BEGIN
	// =============================================================================================================================
	// Purpose: Reditech standard typical for controlling a digital valve (open/close OR 3-way valve)
	// -----------------------------------------------------------------------------------------------------------------------------
	// Date (dd MMM yyyy)   Developer                                   Version Comments/Reason for change
	// ..................   .........                                   ....... ..........................
	// 10 Dec 2018          Bram Verheyen                               08.0    Full review
	// 30 Jan 2019          Matthias De Staelen                         08.1    Outputs can be high in simulation mode
	// =============================================================================================================================

	//============================================================================================
	#b_CfgEnOutpAlwaysOn := #Iw_Cfg.%X1;
	#b_CfgEnFbPos1 := #Iw_Cfg.%X2;
	#b_CfgEnFbPos0 := #Iw_Cfg.%X3;
	#b_CfgSafPosPos1 := #Iw_Cfg.%X4;
	#b_CfgPushToRun := #Iw_Cfg.%X8;
	#b_CfgDisableSim := #Iw_Cfg.%X10;
	#b_CfgStopArea := #Iw_Cfg.%X11;

	//============================================================================================
	#b_DisAlmWrn := #Ib_DisAlmWrn OR #IO_AreaCmd.Alm.Dis OR #b_StaModDis;

	//============================================================================================
	#b_StaSaf := (#Iby_Saf <> 0) AND NOT #b_DisAlmWrn;
	#b_StaIlOn := (#Iby_IlOn <> 0);
	#b_StaIlOff := (#Iby_IlOff <> 0);

	//============================================================================================
	#b_HmiCmdModAut := #IOdi_HmiCmd.%X0;
	#b_HmiCmdModMan := #IOdi_HmiCmd.%X1;
	#b_HmiCmdModDis := #IOdi_HmiCmd.%X2;
	#b_HmiCmdSim := #IOdi_HmiCmd.%X3;
	#b_HmiCmdPos1 := #IOdi_HmiCmd.%X4;
	#b_HmiCmdPos0 := #IOdi_HmiCmd.%X5;
	#b_HmiCmdStp := #IOdi_HmiCmd.%X6;
	#b_HmiCmdRst := #IOdi_HmiCmd.%X7;
	#b_HmiCmdRstActCou := #IOdi_HmiCmd.%X8;

	IF #b_CfgPushToRun THEN
	    #IOdi_HmiCmd := DWORD_TO_DINT(DINT_TO_DWORD(#IOdi_HmiCmd) AND 48);
	ELSE
	    #IOdi_HmiCmd := 0;
	END_IF;

	//============================================================================================
	IF #IO_AreaCmd.Mode.AreaMode THEN
	    #b_ReqAut := #IO_AreaCmd.Mode.Auto;
	    #b_ReqMan := #IO_AreaCmd.Mode.Man;
	    #b_ReqDis := #IO_AreaCmd.Mode.Dis;
	ELSE
	    #b_ReqAut := #b_HmiCmdModAut;
	    #b_ReqMan := #b_HmiCmdModMan;
	    #b_ReqDis := #b_HmiCmdModDis;
	END_IF;

	IF (#b_ReqAut AND NOT #b_ReqMan AND NOT #b_ReqDis) THEN
	    #b_StaModAut := true;
	    #b_StaModMan := false;
	    #b_StaModDis := false;
	END_IF;
	IF (#b_ReqMan AND NOT #b_ReqAut AND NOT #b_ReqDis) THEN
	    #b_StaModAut := false;
	    #b_StaModMan := true;
	    #b_StaModDis := false;
	END_IF;
	IF (#b_ReqDis AND NOT #b_ReqAut AND NOT #b_ReqMan) THEN
	    #b_StaModAut := false;
	    #b_StaModMan := false;
	    #b_StaModDis := true;
	END_IF;

	//============================================================================================
	IF #IO_AreaCmd.Sim.ForceOn OR (#b_HmiCmdSim AND NOT #b_StaSim AND NOT #IO_AreaCmd.Sim.ForceOn AND NOT #IO_AreaCmd.Sim.ForceOff) THEN
	    #b_StaSim := true;
	    #b_HmiCmdSim := false; // reset of command necessary, else simulation will always be reset immediately by following instructions
	END_IF;
	IF #IO_AreaCmd.Sim.ForceOff OR (#b_HmiCmdSim AND #b_StaSim AND NOT #IO_AreaCmd.Sim.ForceOn AND NOT #IO_AreaCmd.Sim.ForceOff) THEN
	    #b_StaSim := false;
	    #b_HmiCmdSim := false;
	END_IF;

	//============================================================================================
	#b_AlActCtn := #Iby_CfgActionAlm.%X0;
	#b_AlActSaf := #Iby_CfgActionAlm.%X1;
	#b_AlActStp := #Iby_CfgActionAlm.%X2;

	#b_CfgAlmActCtn := #b_AlActCtn OR (NOT #b_AlActCtn AND NOT #b_AlActSaf AND NOT #b_AlActStp);
	#b_CfgAlmActSaf := (NOT #b_AlActCtn AND #b_AlActSaf);
	#b_CfgAlmActStp := (NOT #b_AlActCtn AND NOT #b_AlActSaf AND #b_AlActStp);

	//============================================================================================
	IF (#b_ReqPos1 AND NOT #b_FbSimPos1) OR (#b_ReqPos0 AND NOT #b_FbSimPos0) THEN
	    #b_FbSimPos1 := false;
	    #b_FbSimPos0 := false;
	END_IF;
	IF ((#i_TmrFbPos1 <= 1) OR #Ii_ParTFb = 0) AND #b_ReqPos1 THEN
	    #b_FbSimPos1 := true;
	    #b_FbSimPos0 := false;
	END_IF;
	IF ((#i_TmrFbPos0 <= 1) OR #Ii_ParTFb = 0) AND #b_ReqPos0 THEN
	    #b_FbSimPos1 := false;
	    #b_FbSimPos0 := true;
	END_IF;

	//============================================================================================
	#Ob_StaPos1 := (#b_CfgEnFbPos1 AND #Ib_FbPos1 AND NOT #b_StaSim)
	OR (NOT #b_CfgEnFbPos1 AND #b_FbSimPos1)
	OR (#b_StaSim AND #b_FbSimPos1);
	#Ob_StaPos0 := (#b_CfgEnFbPos0 AND #Ib_FbPos0 AND NOT #b_StaSim)
	OR (NOT #b_CfgEnFbPos0 AND #b_FbSimPos0)
	OR (#b_StaSim AND #b_FbSimPos0);

	//============================================================================================
	#b_NoAlm := false;
	#b_RstAlm := #b_HmiCmdRst OR #IO_AreaCmd.Alm.Rst;
	"FC_UTIL_AlmAck"(Ib_CmdAck := #b_RstAlm,
	                 Oi_StaAlm => #i_dummy,
	                 Ob_StaAlm => #b_dummy,
	                 Ob_StaNewAlm => #b_StaAlmNew,
	                 IO_Alm0 := #b_AlmToFb,
	                 IO_Alm1 := #b_AlmIncFb,
	                 IO_Alm2 := #b_AlmIncIl,
	                 IO_Alm3 := #b_NoAlm,
	                 IO_Alm4 := #b_NoAlm,
	                 IO_Alm5 := #b_NoAlm,
	                 IO_Alm6 := #b_NoAlm,
	                 IO_Alm7 := #b_NoAlm,
	                 IO_Alm8 := #b_NoAlm,
	                 IO_Alm9 := #b_NoAlm,
	                 IO_Alm10 := #b_NoAlm,
	                 IO_Alm11 := #b_NoAlm,
	                 IO_Alm12 := #b_NoAlm,
	                 IO_Alm13 := #b_NoAlm,
	                 IO_Alm14 := #b_NoAlm,
	                 IO_Alm15 := #b_NoAlm,
	                 IOi_StaAck := #i_AlmAck);

	//============================================================================================
	IF (#Ii_ParTFb > 0) THEN  // only when time value > 0
	    #FB_UTIL_TON_Del_1(Ii_tValue := #Ii_ParTFb,
	                       Ib_In := (#b_ReqPos1 AND NOT #Ob_StaPos1),
	                       Ii_Base := 1,
	                       Ib_Hold := 0,
	                       Ob_Out => #b_FbErrPos1,
	                       Oi_tmrValue => #i_TmrFbPos1);
	END_IF;

	IF (#Ii_ParTFb > 0) THEN  // only when time value > 0
	    #FB_UTIL_TON_Del_2(Ii_tValue := #Ii_ParTFb,
	                       Ib_In := (#b_ReqPos0 AND NOT #Ob_StaPos0),
	                       Ii_Base := 1,
	                       Ib_Hold := 0,
	                       Ob_Out => #b_FbErrPos0,
	                       Oi_tmrValue => #i_TmrFbPos0);
	END_IF;

	IF ((#b_FbErrPos0 OR #b_FbErrPos1) AND (#Ii_ParTFb > 0)) AND NOT #b_DisAlmWrn THEN
	    #b_AlmToFb := true;
	END_IF;

	//============================================================================================
	IF (#Ii_ParTFb > 0) THEN  // only when time value > 0
	    #FB_UTIL_TON_Del_3(Ii_tValue := #Ii_ParTFb,
	                       Ib_In := (#Ob_StaPos1 AND #Ob_StaPos0),
	                       Ii_Base := 1,
	                       Ib_Hold := 0,
	                       Ob_Out => #b_IncFbErr,
	                       Oi_tmrValue => #i_TmrIncFb);
	END_IF;

	IF (#Ob_StaPos1 AND #Ob_StaPos0 AND #b_IncFbErr) AND NOT #b_DisAlmWrn THEN
	    #b_AlmIncFb := true;
	END_IF;

	//============================================================================================
	IF (#b_StaIlOn AND #b_StaIlOff) AND NOT #b_DisAlmWrn THEN
	    #b_AlmIncIl := true;
	END_IF;
	IF NOT (#b_StaIlOn AND #b_StaIlOff) THEN
	    #b_AlmIncIl := false;
	END_IF;

	//============================================================================================
	#b_StaAlm := #b_AlmToFb OR #b_StaSaf OR #b_AlmIncFb OR #b_AlmIncIl;
	#Ob_Alm := #b_StaAlm;

	//============================================================================================
	#b_CmdAutPos1 := #Ib_AutPos1;
	#b_CmdAutPos0 := #Ib_AutPos0;

	IF #b_StaModAut THEN
	    #b_CmdManPos1 := #b_CmdAutPos1;
	    #b_CmdManPos0 := #b_CmdAutPos0;
	END_IF;

	//============================================================================================
	IF #b_StaModMan AND NOT #b_CfgPushToRun THEN
	    IF (#b_HmiCmdPos1 OR (#b_StaSaf AND #b_CfgSafPosPos1) OR (#b_AlmToFb AND #b_CfgAlmActSaf AND #b_CfgSafPosPos1)) THEN
	        #b_CmdManPos1 := true;
	        #b_CmdManPos0 := false;
	    END_IF;
	    IF (#b_HmiCmdPos0 OR (#b_StaSaf AND NOT #b_CfgSafPosPos1) OR (#b_AlmToFb AND #b_CfgAlmActSaf AND NOT #b_CfgSafPosPos1)) THEN
	        #b_CmdManPos1 := false;
	        #b_CmdManPos0 := true;
	    END_IF;
	    IF #b_HmiCmdStp OR #b_StaAlm OR #b_StaModDis THEN
	        #b_CmdManPos1 := false;
	        #b_CmdManPos0 := false;
	    END_IF;
	END_IF;

	IF #b_StaModMan AND #b_CfgPushToRun THEN
	    #b_CmdManPos1 := ((#b_HmiCmdPos1 AND NOT #b_HmiCmdPos0)
	    OR (#b_StaSaf AND #b_CfgSafPosPos1)
	    OR (#b_AlmToFb AND #b_CfgAlmActSaf AND #b_CfgSafPosPos1)) AND NOT (#b_AlmToFb AND #b_CfgAlmActStp)
	    AND NOT #b_StaModDis;
	    #b_CmdManPos0 := ((#b_HmiCmdPos0 AND NOT #b_HmiCmdPos1)
	    OR (#b_StaSaf AND NOT #b_CfgSafPosPos1)
	    OR (#b_AlmToFb AND #b_CfgAlmActSaf AND NOT #b_CfgSafPosPos1)) AND NOT (#b_AlmToFb AND #b_CfgAlmActStp)
	    AND NOT #b_StaModDis;
	END_IF;

	IF NOT #b_StaModMan OR #b_StaModDis THEN
	    #b_CmdManPos1 := false;
	    #b_CmdManPos0 := false;
	END_IF;




	//============================================================================================
	#b_CmdPos1 := (#b_StaModAut AND #b_CmdAutPos1) OR (#b_StaModMan AND #b_CmdManPos1);
	#b_CmdPos0 := (#b_StaModAut AND #b_CmdAutPos0) OR (#b_StaModMan AND #b_CmdManPos0);

	//============================================================================================
	#b_ReqOutPos1 := (#b_CmdPos1 AND NOT #b_StaAlm AND NOT #b_StaIlOn)
	OR (#b_CmdPos1 AND #b_StaAlm AND NOT #b_StaSaf AND #b_CfgAlmActCtn)
	OR (#b_StaIlOff AND NOT #b_StaAlm AND NOT #b_StaIlOn)
	OR (#b_StaSaf AND #b_CfgSafPosPos1)
	OR (#b_AlmToFb AND #b_CfgAlmActSaf AND #b_CfgSafPosPos1);

	#b_ReqOutPos0 := (#b_CmdPos0 AND NOT #b_StaAlm AND NOT #b_StaIlOff)
	OR (#b_CmdPos0 AND #b_StaAlm AND NOT #b_StaSaf AND #b_CfgAlmActCtn)
	OR (#b_StaIlOn AND NOT #b_StaAlm AND NOT #b_StaIlOff)
	OR (#b_StaSaf AND NOT #b_CfgSafPosPos1)
	OR (#b_AlmToFb AND #b_CfgAlmActSaf AND NOT #b_CfgSafPosPos1);

	#b_ReqPos1 := (#b_ReqOutPos1 AND #b_CfgEnOutpAlwaysOn)
	OR (#b_ReqOutPos1 AND NOT #b_CfgEnOutpAlwaysOn AND NOT #Ob_StaPos1)
	AND NOT #b_StaModDis;
	#b_ReqPos0 := (#b_ReqOutPos0 AND #b_CfgEnOutpAlwaysOn)
	OR (#b_ReqOutPos0 AND NOT #b_CfgEnOutpAlwaysOn AND NOT #Ob_StaPos0)
	AND NOT #b_StaModDis;

	//============================================================================================
	#Ob_Pos0 := #b_ReqPos0;
	#Ob_Pos1 := #b_ReqPos1;
	#Ob_Stp := NOT #Ob_Pos0 AND NOT #Ob_Pos1;

	//============================================================================================
	#Odi_HmiSta.%X0 := #b_StaModAut;
	#Odi_HmiSta.%X1 := #b_StaModMan;
	#Odi_HmiSta.%X2 := #b_StaModDis;
	#Odi_HmiSta.%X3 := #b_StaSim;
	#Odi_HmiSta.%X4 := #b_StaIlOff;
	#Odi_HmiSta.%X5 := #b_StaIlOn;
	#Odi_HmiSta.%X6 := #b_StaSaf;
	#Odi_HmiSta.%X16 := #b_ReqPos1;
	#Odi_HmiSta.%X17 := #b_ReqPos0;
	#Odi_HmiSta.%X18 := #Ob_StaPos1 AND NOT #b_StaAlm;
	#Odi_HmiSta.%X19 := #Ob_StaPos0 AND NOT #b_StaAlm;
	#Odi_HmiSta.%X20 := #b_StaAlm;
	#Odi_HmiSta.%X28 := #IO_AreaCmd.Mode.AreaMode;
	#Odi_HmiSta.%X29 := #b_CfgAlmActCtn;
	#Odi_HmiSta.%X30 := #b_CfgAlmActSaf;
	#Odi_HmiSta.%X31 := #b_CfgAlmActStp;

	#Oi_HMIStaInd.%X0 := 0;
	#Oi_HMIStaInd.%X0 := #b_StaModAut;
	#Oi_HMIStaInd.%X1 := #b_StaModMan;
	#Oi_HMIStaInd.%X2 := #b_StaModDis;
	#Oi_HMIStaInd.%X3 := #b_StaSim;
	#Oi_HMIStaInd.%X4 := #b_StaAlm;
	#Oi_HMIStaInd.%X5 := #Ob_StaPos1 AND NOT #b_StaAlm;
	#Oi_HMIStaInd.%X6 := #Ob_StaPos0 AND NOT #b_StaAlm;

	#I_HmiSta.%X0 := #b_StaModAut;
	#I_HmiSta.%X1 := #b_StaModMan;
	#I_HmiSta.%X2 := #b_StaModDis;
	#I_HmiSta.%X3 := #b_StaSim;
	#I_HmiSta.%X4 := #b_StaIlOn;
	#I_HmiSta.%X5 := #b_StaIlOff;
	#I_HmiSta.%X6 := #Ob_StaPos1;
	#I_HmiSta.%X7 := #Ob_StaPos0;
	#I_HmiSta.%X8 := #b_StaAlm;

	//============================================================================================
	#di_AUX := 0;
	#di_AUX.%X0 := #b_AlmToFb;
	#di_AUX.%X1 := #b_AlmIncFb;
	#di_AUX.%X2 := #b_AlmIncIl;
	#di_AUX.%X8 := #Iby_IlOff.%X0;
	#di_AUX.%X9 := #Iby_IlOff.%X1;
	#di_AUX.%X10 := #Iby_IlOff.%X2;
	#di_AUX.%X11 := #Iby_IlOff.%X3;
	#di_AUX.%X12 := #Iby_IlOff.%X4;
	#di_AUX.%X13 := #Iby_IlOff.%X5;
	#di_AUX.%X14 := #Iby_IlOff.%X6;
	#di_AUX.%X15 := #Iby_IlOff.%X7;
	#di_AUX.%X16 := #Iby_IlOn.%X0;
	#di_AUX.%X17 := #Iby_IlOn.%X1;
	#di_AUX.%X18 := #Iby_IlOn.%X2;
	#di_AUX.%X19 := #Iby_IlOn.%X3;
	#di_AUX.%X20 := #Iby_IlOn.%X4;
	#di_AUX.%X21 := #Iby_IlOn.%X5;
	#di_AUX.%X22 := #Iby_IlOn.%X6;
	#di_AUX.%X23 := #Iby_IlOn.%X7;
	#di_AUX.%X24 := #Iby_Saf.%X0;
	#di_AUX.%X25 := #Iby_Saf.%X1;
	#di_AUX.%X26 := #Iby_Saf.%X2;
	#di_AUX.%X27 := #Iby_Saf.%X3;
	#di_AUX.%X28 := #Iby_Saf.%X4;
	#di_AUX.%X29 := #Iby_Saf.%X5;
	#di_AUX.%X30 := #Iby_Saf.%X6;
	#di_AUX.%X31 := #Iby_Saf.%X7;
	#Odi_HmiAlm := #di_AUX;

	//============================================================================================
	#di_AUX := 0;
	#di_AUX.%X0 := #b_AlmToFb;
	#di_AUX.%X1 := #b_AlmIncFb;
	#di_AUX.%X2 := #b_AlmIncIl;
	#Oi_HmiAlm := DINT_TO_INT(#di_AUX);

	//============================================================================================
	IF #b_StaModDis THEN
	    #IO_AreaFb.Mode.Dis := TRUE;
	END_IF;
	IF #b_StaModMan THEN
	    #IO_AreaFb.Mode.Man := TRUE;
	END_IF;
	IF #b_StaModAut THEN
	    #IO_AreaFb.Mode.Auto := TRUE;
	END_IF;
	IF #b_StaAlm THEN
	    #IO_AreaFb.Alm.Alm := TRUE;
	END_IF;
	IF #b_StaAlmNew THEN
	    #IO_AreaFb.Alm.New := TRUE;
	END_IF;
	IF #b_StaAlm AND #b_CfgStopArea THEN
	    #IO_AreaFb.Alm.StopArea := TRUE;
	END_IF;
	IF #b_StaSim THEN
	    #IO_AreaFb.Sim.Sim := TRUE;
	END_IF;

	//Generating alarm category feedback
	IF #i_Category = 1 AND #b_StaAlm THEN
	    #IO_AreaFb.Alm.Alm_Lvl1 := TRUE;
	END_IF;

	IF #i_Category = 2 AND #b_StaAlm THEN
	    #IO_AreaFb.Alm.Alm_Lvl2 := TRUE;
	END_IF;

	IF #i_Category = 3 AND #b_StaAlm THEN
	    #IO_AreaFb.Alm.Alm_Lvl3 := TRUE;
	END_IF;

	//============================================================================================
	IF (#Ob_Pos0 AND NOT #b_Old_Ob_Pos0) OR (#Ob_Pos1 AND NOT #b_Old_Ob_Pos1) THEN
	    #Odi_ActCouRst := #Odi_ActCouRst + 1;
	    #Odi_ActCouTot := #Odi_ActCouTot + 1;
	END_IF;
	IF #b_HmiCmdRstActCou THEN
	    #Odi_ActCouRst := 0;
	END_IF;
	#b_Old_Ob_Pos0 := #Ob_Pos0;
	#b_Old_Ob_Pos1 := #Ob_Pos1;
END_FUNCTION_BLOCK

FUNCTION_BLOCK "FB_CM_DI"
TITLE = Digital input
{ S7_Optimized_Access := 'FALSE' }
AUTHOR : Reditech
FAMILY : Typical
VERSION : 0.0
//Reditech standard typical for controlling a digital input (switch) inversion is possible, input is delayed
   VAR_INPUT
      Ib_InRaw : Bool;   //  digital input
      Ib_Inv : Bool;   //  invert digital input
      Ii_ParTOn : Int;   //  time delay value ON
      Ii_ParTOff : Int;   //  time delay value OFF
      Ib_EnAlmIfzero : Bool;
      Ib_EnAlmIfOne : Bool;
      Ib_EnWrnIfzero : Bool;
      Ib_EnWrnIfOne : Bool;
      Ib_DisAlmWrn : Bool;
      Iw_Cfg : Word;   //  .0=alarm if out = 0 / .1=alarm if out = 1 / .2=automatic alarm reset / .4 = warning if out =0 / .5 = warning if out =1
   END_VAR

   VAR_OUTPUT
      Ob_Out : Bool;   //  Output value
      Ob_Alm : Bool;   //  general alarm
      Ob_Wrn : Bool;   //  general warning
      Odi_HmiSta : DInt;   //  State bits for HMI
      Odi_HmiAlm : DInt;   //  Alarm bit for HMI
      Oi_HmiAlm : Int;   //  Alarm bit for HMI
   END_VAR

   VAR_IN_OUT
      IOdi_HmiCmd : DInt;   //  Command bits from HMI
      IO_AreaCmd : "UDT_AreaCmd";   //  Command bits from area
      IO_AreaFb : "UDT_AreaFb";   //  Feedback bits to area
   END_VAR

   VAR
      i_TmrOn { ExternalVisible := 'False'} : Int;   //  actual timer value delay ON
      i_TmrOff { ExternalVisible := 'False'} : Int;   //  actual timer value delay OFF
      b_HmiCmdSim { ExternalVisible := 'False'} : Bool;   //  command (toggle) simulation mode
      b_HmiCmdSimValOn { ExternalVisible := 'False'} : Bool;   //  set simulation value on
      b_HmiCmdSimValOff { ExternalVisible := 'False'} : Bool;   //  set simulation value off
      b_HmiCmdRst { ExternalVisible := 'False'} : Bool;   //  reset alarm
      b_StaSim { ExternalVisible := 'False'} : Bool;   //  simulation mode on
      b_StaInRaw { ExternalVisible := 'False'} : Bool;   //  copy of input value
      b_StaAlm { ExternalVisible := 'False'} : Bool;   //  alarm
      b_StaOut { ExternalVisible := 'False'} : Bool;   //  output
      b_StaWrn { ExternalVisible := 'False'} : Bool;   //  warning
      b_CfgAutoReset { ExternalVisible := 'False'} : Bool;   //  automatic alarm reset
      b_CfgStopArea { ExternalVisible := 'False'} : Bool;
      b_Alm { ExternalVisible := 'False'} : Bool;   //  alarm
      b_Wrn { ExternalVisible := 'False'} : Bool;   //  warning
      b_In { ExternalVisible := 'False'} : Bool;   //  auxiliary bit for input value before delays
      b_TOnOut { ExternalVisible := 'False'} : Bool;   //  time delay ON finished
      b_TOffOut { ExternalVisible := 'False'} : Bool;   //  time delay OFF finished
      Fb_UTIL_Ton_Del { ExternalVisible := 'False'} : "FB_UTIL_TON_Sec";
      FB_UTIL_TOF_Del { ExternalVisible := 'False'} : "FB_UTIL_TON_Sec";
      b_DisAlmWrn : Bool;
      b_dummy : Bool;
      i_dummy : Int;
      b_StaAlmNew : Bool;
      b_NoAlm : Bool;
      i_AlmAck : Int;
      b_DisAlmWrn_1 : Bool;
      b_RstAlm : Bool;
      i_Category : Int;   // Device alarm category setting
   END_VAR

   VAR_TEMP
      di_AUX : DInt;   //  auxiliary double word for calculation of state or alarm word to HMI
   END_VAR


BEGIN
	// =========================================================================================================================
	// Purpose: Reditech standard typical for controlling a digital input (switch) inversion is possible, input is delayed
	// -------------------------------------------------------------------------------------------------------------------------
	// Date (dd MMM yyyy)   Developer                                   Version Comments/Reason for change
	// ..................   .........                                   ....... ..........................
	// 18 Dec 2018          Bram Verheyen                               09.0    Full review
	// =========================================================================================================================

	//============================================================================================
	#b_CfgAutoReset := #Iw_Cfg.%X2;
	#b_CfgStopArea := #Iw_Cfg.%X11;

	//============================================================================================
	#b_DisAlmWrn := #Ib_DisAlmWrn OR #IO_AreaCmd.Alm.Dis;

	//============================================================================================
	#b_HmiCmdSim := #IOdi_HmiCmd.%X0;
	#b_HmiCmdSimValOn := #IOdi_HmiCmd.%X1;
	#b_HmiCmdSimValOff := #IOdi_HmiCmd.%X2;
	#b_HmiCmdRst := #IOdi_HmiCmd.%X3;
	#IOdi_HmiCmd := 0;

	//============================================================================================
	IF #IO_AreaCmd.Sim.ForceOn OR (#b_HmiCmdSim AND NOT #b_StaSim AND NOT #IO_AreaCmd.Sim.ForceOn AND NOT #IO_AreaCmd.Sim.ForceOff) THEN
	    #b_StaSim := true;
	    #b_HmiCmdSim := false; // reset of command necessary, else simulation will always be reset immediately by following instructions
	END_IF;
	IF #IO_AreaCmd.Sim.ForceOff OR (#b_HmiCmdSim AND #b_StaSim AND NOT #IO_AreaCmd.Sim.ForceOn AND NOT #IO_AreaCmd.Sim.ForceOff) THEN
	    #b_StaSim := false;
	    #b_HmiCmdSim := false;
	END_IF;

	//============================================================================================
	IF NOT #b_StaSim THEN
	    IF NOT #Ib_Inv THEN
	        #b_In := #Ib_InRaw;
	    ELSE
	        #b_In := NOT #Ib_InRaw;
	    END_IF;
	    #b_StaInRaw := #Ib_InRaw;
	ELSE
	    IF #b_HmiCmdSimValOn THEN
	        #b_In := true;
	    END_IF;
	    IF #b_HmiCmdSimValOff THEN
	        #b_In := false;
	    END_IF;
	    #b_StaInRaw := #b_In;
	END_IF;

	//============================================================================================
	#Fb_UTIL_Ton_Del(Ii_tValue := #Ii_ParTOn,
	                 Ib_In := #b_In AND (#Ib_EnAlmIfOne OR #Ib_EnWrnIfOne) AND NOT #b_DisAlmWrn,
	                 Ii_Base := 1,
	                 Ib_Hold := 0,
	                 Ob_Out => #b_TOnOut,
	                 Oi_tmrValue => #i_TmrOn);

	#FB_UTIL_TOF_Del(Ii_tValue := #Ii_ParTOff,
	                 Ib_In := (NOT #b_In AND (#Ib_EnAlmIfzero OR #Ib_EnWrnIfzero) AND NOT #b_DisAlmWrn),
	                 Ii_Base := 1,
	                 Ib_Hold := 0,
	                 Ob_Out => #b_TOffOut,
	                 Oi_tmrValue => #i_TmrOff);

	#b_StaOut := #b_In;
	//============================================================================================
	#b_NoAlm := false;
	#b_RstAlm := #b_HmiCmdRst OR #IO_AreaCmd.Alm.Rst OR #b_CfgAutoReset;
	"FC_UTIL_AlmAck"(Ib_CmdAck := #b_RstAlm,
	                 Oi_StaAlm => #i_dummy,
	                 Ob_StaAlm => #b_dummy,
	                 Ob_StaNewAlm => #b_StaAlmNew,
	                 IO_Alm0 := #b_Alm,
	                 IO_Alm1 := #b_Wrn,
	                 IO_Alm2 := #b_NoAlm,
	                 IO_Alm3 := #b_NoAlm,
	                 IO_Alm4 := #b_NoAlm,
	                 IO_Alm5 := #b_NoAlm,
	                 IO_Alm6 := #b_NoAlm,
	                 IO_Alm7 := #b_NoAlm,
	                 IO_Alm8 := #b_NoAlm,
	                 IO_Alm9 := #b_NoAlm,
	                 IO_Alm10 := #b_NoAlm,
	                 IO_Alm11 := #b_NoAlm,
	                 IO_Alm12 := #b_NoAlm,
	                 IO_Alm13 := #b_NoAlm,
	                 IO_Alm14 := #b_NoAlm,
	                 IO_Alm15 := #b_NoAlm,
	                 IOi_StaAck := #i_AlmAck);

	//============================================================================================
	IF ((#b_TOnOut AND #Ib_EnAlmIfOne) OR (#b_TOffOut AND #Ib_EnAlmIfzero)) AND NOT #b_DisAlmWrn THEN
	    #b_Alm := true;

	END_IF;

	//============================================================================================
	IF ((#b_TOnOut AND #Ib_EnWrnIfOne) OR (#b_TOffOut AND #Ib_EnWrnIfzero)) AND NOT #b_DisAlmWrn THEN
	    #b_Wrn := true;
	END_IF;

	//============================================================================================
	#b_StaAlm := #b_Alm;
	#Ob_Alm := #b_Alm;

	//============================================================================================
	#b_StaWrn := #b_Wrn;
	#Ob_Wrn := #b_Wrn;

	//============================================================================================
	#Ob_Out := #b_StaOut;

	//============================================================================================
	#Odi_HmiSta.%X0 := #b_StaSim;
	#Odi_HmiSta.%X1 := #b_StaInRaw;
	#Odi_HmiSta.%X16 := #b_StaAlm;
	#Odi_HmiSta.%X17 := #b_StaOut;
	#Odi_HmiSta.%X18 := #b_StaWrn;
	#Odi_HmiSta.%X28 := #IO_AreaCmd.Mode.AreaMode;

	//Sending data to HMI for animated alarm category
	#Odi_HmiSta.%X8 := #i_Category = 1 AND #b_StaAlm;
	#Odi_HmiSta.%X9 := #i_Category = 2 AND #b_StaAlm;
	#Odi_HmiSta.%X19 := #i_Category = 3 AND #b_StaAlm;

	//============================================================================================
	#di_AUX := 0;
	#di_AUX.%X0 := #b_Alm;
	#di_AUX.%X1 := #b_Wrn;
	#Odi_HmiAlm := #di_AUX;
	#Oi_HmiAlm := DINT_TO_INT(#Odi_HmiAlm);

	//============================================================================================
	IF #b_StaAlm THEN
	    #IO_AreaFb.Alm.Alm := TRUE;
	END_IF;
	IF #b_StaWrn THEN
	    #IO_AreaFb.Alm.Wrn := TRUE;
	END_IF;
	IF #b_StaSim THEN
	    #IO_AreaFb.Sim.Sim := TRUE;
	END_IF;
	IF #b_StaAlmNew THEN
	    #IO_AreaFb.Alm.New := TRUE;
	END_IF;
	IF #b_StaAlm AND #b_CfgStopArea THEN
	    #IO_AreaFb.Alm.StopArea := TRUE;
	END_IF;

	//Generating alarm category feedback
	IF #i_Category = 1 AND #b_StaAlm THEN
	    #IO_AreaFb.Alm.Alm_Lvl1 := TRUE;
	END_IF;

	IF #i_Category = 2 AND #b_StaAlm THEN
	    #IO_AreaFb.Alm.Alm_Lvl2 := TRUE;
	END_IF;

	IF #i_Category = 3 AND #b_StaAlm THEN
	    #IO_AreaFb.Alm.Alm_Lvl3 := TRUE;
	END_IF;
END_FUNCTION_BLOCK

FUNCTION_BLOCK "FB_EM_Lvl"
{ S7_Optimized_Access := 'FALSE' }
VERSION : 0.1
   VAR_INPUT
      Ib_RequestEqp { ExternalVisible := 'False'} : Bool;   //  Request equipment Command
      Ib_LvlOff_FirstEqp : Bool;   //  Level switch low low
      Ib_LvlOff_SecondEqp : Bool;   //  Level switch low
      Ib_LvlOn_FirstEqp : Bool;   //  Level switch high
      Ib_LvlOn_SecondEqp : Bool;   //  Level switch High High
      Ib_NrEqp : Bool;   //  Number of equipment used at the same time, 0 = 1 eqp, 1 = 2 eqp
   END_VAR

   VAR_OUTPUT
      Ob_ReqFirstEqp : Bool;   //  Request first equipment
      Ob_ReqSecondEqp : Bool;   //  Request second equipment
   END_VAR

   VAR_IN_OUT
      IO_AreaCmd : "UDT_AreaCmd";   //  Command bits from area
      IO_AreaFb : "UDT_AreaFb";   //  Feedback bits to area
   END_VAR

   VAR
      b_FirstEqpReq : Bool;   //  Request to Equipment 1
      b_SecondEqpReq : Bool;   //  Request to Equipment 2
      b_ReqAut : Bool;   //  Request automatic mode
      b_ReqMan : Bool;
      b_ReqDis : Bool;
   END_VAR


BEGIN
	//not used// =========================================================================================================================
	// Purpose: Reditech standard typical for controlling Pump Toggle manual automatic or semi-automatic
	// -------------------------------------------------------------------------------------------------------------------------
	// Date (dd MMM yyyy)   Developer                                   Version Comments/Reason for change
	// ..................   .........                                   ....... ..........................
	// 16 OCT 2018          Robin Cardinaels                               01      Initial (creation)

	// =========================================================================================================================
	// copy command bits from HMI and reset

	#b_ReqAut := #IO_AreaCmd.Mode.Auto;
	#b_ReqMan := #IO_AreaCmd.Mode.Man;
	#b_ReqDis := #IO_AreaCmd.Mode.Dis;

	IF NOT #b_ReqAut THEN
	    #b_FirstEqpReq := #b_SecondEqpReq := false;
	ELSE
	    IF #Ib_LvlOn_FirstEqp THEN
	        #b_FirstEqpReq := TRUE;
	    END_IF;
	    IF #Ib_LvlOff_FirstEqp THEN
	        #b_FirstEqpReq := FALSE;
	    END_IF;

	    IF #Ib_NrEqp THEN
	        // setting control bits for anaog and digital control.
	        IF #Ib_LvlOn_SecondEqp THEN
	            #b_SecondEqpReq := TRUE;
	        END_IF;
	        IF #Ib_LvlOff_SecondEqp THEN
	            #b_SecondEqpReq := FALSE;
	        END_IF;
	    ELSE
	        #b_SecondEqpReq := false;
	    END_IF;
	END_IF;

	// Set Output For Motor 1
	#Ob_ReqFirstEqp := #Ib_RequestEqp AND #b_FirstEqpReq;

	//Set output for Motor 2
	#Ob_ReqSecondEqp := #Ib_RequestEqp AND #b_SecondEqpReq;

END_FUNCTION_BLOCK

FUNCTION_BLOCK "FB_EM_Toggle_2Eqp"
{ S7_Optimized_Access := 'FALSE' }
VERSION : 0.1
   VAR_INPUT
      Ib_RequestEqp : Bool;   //  Request equipment Command
      Ib_RequestCompEqp : Bool;   //  Request complementary equipment Command
      Ib_ExtToggle : Bool;   //  External Manual toggle
      Ib_Eqp1Fb : Bool;   //  Equipment 1 Running / Open
      Ib_Eqp1Error : Bool;   //  Equipment 1 Error
      Ii_Eqp1OpHours : DInt;   //  Equipment 1 operating hours
      Ib_Eqp2Fb : Bool;   //  Equipment 2 Running / Open
      Ib_Eqp2Error : Bool;   //  Equipment 2 Error
      Ii_Eqp2OpHours : DInt;   //  Equipment 2 Operating hours
      Ii_TBlckStrt : Int;   //  Block simultaniuos Strting time
      Ib_EqpComp : Bool;   //  The equipment complement each other
      Ib_CfgTogRun : Bool;   //  Toggle on running hours
      Ib_EnMan : Bool;   //  Enable manual action
   END_VAR

   VAR_OUTPUT
      Ob_ReqEqp1 : Bool;   //  Request Equipment 1
      Ob_ReqEqp2 : Bool;   //  Request Equipment 2
      Ob_Alm : Bool;   //  General alarm
      Ob_Wrn : Bool;   //  General warning
      Odi_HmiSta : DInt;   //  State bits for HMI
      Odi_HmiAlm : DInt;   //  Alarm bits for HMI
      Oi_HmiAlm : Int;   //  Alarm bits for HMI
   END_VAR

   VAR_IN_OUT
      IOdi_HmiFcnCmd : DInt;   //  .0: automatic/ .1:semiauto/ .2:manual
      IOdi_HmiCmd : DInt;   //  Command bits from HMI
      IO_AreaCmd : "UDT_AreaCmd";   //  Command bits from area
      IO_AreaFb : "UDT_AreaFb";   //  Feedback bits to area
   END_VAR

   VAR
      b_HmiCmdModAut : Bool;   //  HMI Command Automatic mode
      b_HmiCmdRst : Bool;   //  HMI Command Reset
      b_HmiCmdModMan : Bool;   //  HMI Command Manual mode
      b_HmiCmdModDis : Bool;   //  HMI Command disabled Mode
      b_HmiCmdFrcEqp1First : Bool;   //  HMI Command Force equipment 1 first
      b_HmiCmdFrcEqp2First : Bool;   //  HMI Command Force equipment 2 first
      b_HmiFcnCmdAuto : Bool := TRUE;   //  HMI Functional command automatic mode
      b_HmiFcnCmdManual : Bool;   //  HMI Functional command manual mode
      b_HmiStaAlm : Bool;   //  HMI Status alarm
      b_HmiStaModAut : Bool;   //  HMI status Ready
      b_HmiStaModMan : Bool;   //  HMI Status Running
      b_HmiStaModDis : Bool;   //  HMI status Preference Eqp
      b_HmiStaFcnAuto : Bool := TRUE;   //  HMI Status Fuction auto switch enabled
      b_HmiStaFcnMan : Bool;   //  HMI Status Fuction manual switch enabled
      b_HmiStaOff : Bool;   //  HMI Status OFF
      b_HmiStaReady : Bool;   //  HMI Status Ready
      b_HmiStaRunning : Bool;   //  HMI Status Running
      b_HmiStaPref1 : Bool;   //  HMI Status Preferd Eqp 1
      b_HmiStaWrn : Bool;   //  HMI Status equipment not ready
      b_HmiStaPref2 : Bool;   //  HMI Status Preferd Eqp 2
      b_HmiStaAreaMode : Bool;   //  HMI Status Area Mode
      b_HmiAlmAlm : Bool;   //  General Alarm
      b_HmiWrnEquip : Bool;   //  Equipment not available
      b_Eqp2First : Bool;   //  Toggle bit for Equipment selection; 1 = Eqp 2 first, 0 = eqp1 first
      b_Temp1 : Bool;   //  Equipments running for RE
      b_PrevTemp1 : Bool;   //  prev equipments running for RE
      b_Temp2 : Bool;   //  command manual toggle for RE
      b_PrevTemp2 : Bool;   //  prev command manual toggle for RE
      FB_UTIL_TON_Del_1 : "FB_UTIL_TON_Sec";   //  Timer block Strt to prevent simultainious Strting
      b_BlckStrt : Bool;   //  Block Strt to prevent Strting simultainous
      b_helpReady : Bool;   //  Help bit for status ready
      b_ReqAut : Bool;   //  Request automatic mode
      b_ReqMan : Bool;
      b_ReqDis : Bool;
   END_VAR

   VAR_TEMP
      di_AUX : DInt;   //  auxiliary double word for calculation of state or alarm word to HMI
   END_VAR


BEGIN
	//not used// =========================================================================================================================
	// Purpose: Reditech standard typical for controlling Pump Toggle manual automatic or semi-automatic
	// -------------------------------------------------------------------------------------------------------------------------
	// Date (dd MMM yyyy)   Developer                                   Version Comments/Reason for change
	// ..................   .........                                   ....... ..........................
	// 16 OCT 2018          Robin Cardinaels                               01      Initial (creation)
	// 15 Jan 2019          Robin Cardinaels                               02      Review
	// =========================================================================================================================
	// copy command bits from HMI and reset
	#b_HmiCmdModAut := #IOdi_HmiCmd.%X0;
	#b_HmiCmdModMan := #IOdi_HmiCmd.%X1;
	#b_HmiCmdRst := #IOdi_HmiCmd.%X3;


	#IOdi_HmiCmd := 0;

	// Copy of Function Command bits
	#b_HmiFcnCmdAuto := #IOdi_HmiFcnCmd.%X0;
	#b_HmiFcnCmdManual := #IOdi_HmiFcnCmd.%X2;
	#b_HmiCmdFrcEqp1First := #IOdi_HmiFcnCmd.%X4;
	#b_HmiCmdFrcEqp2First := #IOdi_HmiFcnCmd.%X5;
	#IOdi_HmiFcnCmd := 0;

	IF #b_HmiStaAreaMode THEN
	    #b_ReqAut := #IO_AreaCmd.Mode.Auto;
	    #b_ReqMan := #IO_AreaCmd.Mode.Man;
	    #b_ReqDis := #IO_AreaCmd.Mode.Dis;
	ELSE
	    #b_ReqAut := #b_HmiCmdModAut AND NOT #b_HmiStaAlm;
	    #b_ReqMan := #b_HmiCmdModMan OR (#b_HmiStaAlm AND NOT #b_HmiStaModDis);
	    #b_ReqDis := #b_HmiCmdModDis;
	END_IF;

	IF (#b_ReqAut AND NOT #b_ReqMan AND NOT #b_ReqDis) THEN
	    #b_HmiStaModAut := true;
	    #b_HmiStaModMan := false;
	    #b_HmiStaModDis := false;
	END_IF;
	IF (#b_ReqMan AND NOT #b_ReqAut AND NOT #b_ReqDis) THEN
	    #b_HmiStaModAut := false;
	    #b_HmiStaModMan := true;
	    #b_HmiStaModDis := false;
	END_IF;
	IF (#b_ReqDis AND NOT #b_ReqAut AND NOT #b_ReqMan) THEN
	    #b_HmiStaModAut := false;
	    #b_HmiStaModMan := false;
	    #b_HmiStaModDis := true;
	END_IF;

	// copy Function modes to status bits
	IF #b_HmiFcnCmdAuto THEN
	    #b_HmiStaFcnAuto := true;
	    #b_HmiStaFcnMan := false;
	END_IF;
	IF #b_HmiFcnCmdManual AND #Ib_EnMan THEN
	    #b_HmiStaFcnAuto := false;
	    #b_HmiStaFcnMan := true;
	END_IF;

	#b_PrevTemp1 := #b_Temp1;// temperoraty variable to get rising edge
	#b_Temp1 := (#Ob_ReqEqp1) OR (#Ob_ReqEqp2);

	// IF auto mode selected check operating hours every Time both motors are not running
	IF (NOT #b_Temp1 AND #b_PrevTemp1) AND (#b_HmiStaFcnAuto AND NOT #b_HmiStaFcnMan) THEN
	    IF #Ib_CfgTogRun THEN //equipment with the lowest operating hours will Strt if Configurated
	        #b_Eqp2First := #Ii_Eqp2OpHours < #Ii_Eqp1OpHours; // reset toggle if equipment1 operating hours <= equipment2 operating hours
	    ELSE
	        #b_Eqp2First := NOT #b_Eqp2First;
	    END_IF;
	END_IF;
	#b_PrevTemp2 := #b_Temp2; // prev value of manual toggle command for RE
	#b_Temp2 := #Ib_ExtToggle; // manual toggle command
	//toggle equipments if manual toggle requested (hmi or external) and manual toggle configurated
	IF (#b_Temp2 AND NOT #b_PrevTemp2) AND (#b_HmiStaFcnAuto AND NOT #b_HmiStaFcnMan) THEN
	    #b_Eqp2First := NOT #b_Eqp2First;
	END_IF;

	// set equipment 2 actif if equipment 1 not available
	IF (#Ib_Eqp1Error OR #b_HmiCmdFrcEqp2First) AND NOT #Ib_Eqp2Error THEN
	    #b_Eqp2First := TRUE;
	END_IF;
	// set equipment 1 actif if equipment 2 not available
	IF (#Ib_Eqp2Error OR #b_HmiCmdFrcEqp1First) AND NOT #Ib_Eqp1Error THEN
	    #b_Eqp2First := FALSE;
	END_IF;

	// Set Output of FB
	// Set Output For equipment 1
	#Ob_ReqEqp1 := NOT #Ib_Eqp1Error AND (((#Ib_RequestEqp AND NOT #b_Eqp2First) AND (#b_BlckStrt OR #Ob_ReqEqp1) OR (#Ib_RequestCompEqp AND NOT #b_BlckStrt)) AND #Ib_EqpComp)
	OR (NOT #Ib_EqpComp AND #Ib_RequestEqp AND NOT #b_Eqp2First);

	//Set output for equipment 2
	#Ob_ReqEqp2 := NOT #Ib_Eqp2Error AND (((#Ib_RequestEqp AND #b_Eqp2First) AND (#b_BlckStrt OR #Ob_ReqEqp2) OR (#Ib_RequestCompEqp AND NOT #b_BlckStrt)) AND #Ib_EqpComp)
	OR (NOT #Ib_EqpComp AND #Ib_RequestEqp AND #b_Eqp2First);

	// timer to prevent simultanius Strting
	#FB_UTIL_TON_Del_1(Ii_tValue := #Ii_TBlckStrt,
	                   Ib_In := #Ob_ReqEqp1 OR #Ob_ReqEqp2,
	                   Ii_Base := 1,
	                   Ib_Hold := 0);

	// enable starting again
	#b_BlckStrt := NOT #FB_UTIL_TON_Del_1.Ob_Out;

	// HMI Status
	// Status Ready
	#b_helpReady := ((NOT #Ib_Eqp1Error OR NOT #Ib_Eqp2Error) AND NOT #Ib_EqpComp) OR //help bit ready if one equipment availeble in 1+1
	(NOT #Ib_Eqp1Error AND NOT #Ib_Eqp2Error); // or both equipments available
	#b_HmiStaReady := #b_helpReady AND NOT #b_HmiStaRunning;
	//Status Running
	#b_HmiStaRunning := #b_helpReady AND (#Ib_Eqp1Fb OR #Ib_Eqp2Fb);
	//Status OFF
	#b_HmiStaOff := NOT #b_HmiStaReady AND NOT #b_HmiStaRunning;
	// Show Prefferd Pump
	#b_HmiStaPref1 := NOT #b_Eqp2First;
	#b_HmiStaPref2 := #b_Eqp2First;
	//Wrning when motor not available
	#b_HmiWrnEquip := (#Ib_Eqp1Error OR #Ib_Eqp2Error) AND NOT #b_HmiAlmAlm;
	// status warning
	#b_HmiStaWrn := #b_HmiWrnEquip;
	#Ob_Wrn := #b_HmiWrnEquip;
	//Alarm when both pumps ar inavailable // auto reset if equipment is available
	#b_HmiAlmAlm := #Ib_Eqp1Error AND #Ib_Eqp2Error;

	// general alarm
	#b_HmiStaAlm := #b_HmiAlmAlm;
	#Ob_Alm := #b_HmiAlmAlm;

	// copy state bits into double word for HMI
	#di_AUX := 0;

	#di_AUX.%X0 := #b_HmiStaModAut;
	#di_AUX.%X1 := #b_HmiStaModMan;
	#di_AUX.%X2 := #b_HmiStaModDis;
	#di_AUX.%X8 := #b_HmiStaFcnAuto;

	#di_AUX.%X10 := #b_HmiStaFcnMan;
	#di_AUX.%X15 := #b_HmiStaOff;
	#di_AUX.%X16 := #b_HmiStaAlm;
	#di_AUX.%X21 := #b_HmiStaReady;
	#di_AUX.%X22 := #b_HmiStaRunning;
	#di_AUX.%X23 := #b_HmiStaPref1;
	#di_AUX.%X24 := #b_HmiStaWrn;
	#di_AUX.%X25 := #b_HmiStaPref2;
	#di_AUX.%X29 := #b_HmiStaAreaMode;

	#Odi_HmiSta := #di_AUX;

	// copy alarm bits into double word for HMI
	#di_AUX := 0;
	#di_AUX.%X0 := #b_HmiAlmAlm;
	#di_AUX.%X1 := #b_HmiWrnEquip;

	#Odi_HmiAlm := #di_AUX;
	#Oi_HmiAlm := DINT_TO_INT(#di_AUX);

	// Set feedback bits to area
	// #IO_AreaFb.Mode.Dis := #b_HmiStaModDis;
	// #IO_AreaFb.Mode.Man := #b_HmiStaModMan;
	// #IO_AreaFb.Mode.Auto := #b_HmiStaModAut;
	// #IO_AreaFb.Alm.Alm := #b_HmiStaAlm;
	// #IO_AreaFb.Alm.Wrn := #b_HmiStaWrn;
END_FUNCTION_BLOCK

FUNCTION_BLOCK "FB_UM_Mode"
{ S7_Optimized_Access := 'FALSE' }
VERSION : 0.1
   VAR_INPUT
      Ib_CmdRstAlm : Bool;
      Ib_CmdGenRelease : Bool;
      Ib_CmdRstRelease : Bool;
      Ib_CmdGenDis : Bool;
      Ib_AreaStopped : Bool;
      Ib_AreaCmdMode : Bool;
      Ib_SimForceOn : Bool;
      Ib_SimForceOff : Bool;
      Ib_DCSPermissive : Bool;
   END_VAR

   VAR_OUTPUT
      Odi_HmiSta : DInt;
      Ou_AreaCmd : "UDT_AreaCmd";
      Ob_StaExecute : Bool;
      Ob_StaAlm : Bool;
      Ob_StaWrn : Bool;
      Ob_StaRstAlm : Bool;
      Ob_StaSim : Bool;
      Ou_CurrentMode : "UDT_PML_Mode";
   END_VAR

   VAR_IN_OUT
      IOdi_HmiCmd : DInt;
      IOu_AreaFb : "UDT_AreaFb";
      Ib_CmdGenMan : Bool;
      IOw_DCSCmd : Word;
   END_VAR

   VAR
      PML_ModeManager : "FB_PML_ModeManager";
      b_HmiCmdStart : Bool;
      b_HmiCmdModSimOn : Bool;
      b_HmiCmdModMan : Bool;
      b_HmiCmdModDis : Bool;
      b_HmiCmdModAuto : Bool;
      b_HmiCmdRstAlm : Bool;
      b_HmiCmdModSimOff : Bool;
      b_HmiCmdStop : Bool;
      b_StaRun : Bool;
      AreaFb : "UDT_AreaFb";
      AreaCmd : "UDT_AreaCmd";
      b_StaSim { ExternalAccessible := 'False'; ExternalVisible := 'False'; ExternalWritable := 'False'} : Bool;
      StaAreaFb : "UDT_AreaFb";
      b_StaAlm_Lvl1 { S7_SetPoint := 'True'} : Bool;
      b_StaAlm_Lvl2 : Bool;
      b_StaAlm_Lvl3 : Bool;
      I_HmiSta : Word;
   END_VAR


BEGIN
	// =========================================================================================================================
	// Purpose: Reditech standard typical for handling mode transition with the Reditech's standard PackML ModeManager
	// -------------------------------------------------------------------------------------------------------------------------
	// Date (dd MMM yyyy)   Developer                                   Version Comments/Reason for change
	// ..................   .........                                   ....... ..........................
	// 19 NOV 2018          Gijs van Hal                                01      Initial (creation)
	// 20 OCT 2020          Ivan Galhardoni                             02      Implemented manual mode external request input
	// 12 DEC 2020          Ivan Galhardoni                             03      Implemented alarm level animated signaling
	// =========================================================================================================================

	// Copy HMI commands
	#b_HmiCmdModMan := (#IOdi_HmiCmd.%X0 OR (#IOw_DCSCmd.%X1 AND #Ib_DCSPermissive)) OR #Ib_CmdGenMan AND NOT #Ib_CmdGenDis;
	#b_HmiCmdModDis := ((#IOdi_HmiCmd.%X1  OR (#IOw_DCSCmd.%X2 AND #Ib_DCSPermissive)) OR #Ib_CmdGenDis) AND NOT #Ib_CmdGenMan;
	#b_HmiCmdModAuto := (#IOdi_HmiCmd.%X2 OR (#IOw_DCSCmd.%X0 AND #Ib_DCSPermissive)) AND NOT #Ib_CmdGenDis;
	#b_HmiCmdModSimOn := #IOdi_HmiCmd.%X3;
	#b_HmiCmdModSimOff := #IOdi_HmiCmd.%X4;
	#b_HmiCmdStart := (#IOdi_HmiCmd.%X5 OR (#IOw_DCSCmd.%X3 AND #Ib_DCSPermissive)) AND #PML_ModeManager.Ou_ModeCurrent.Production;
	#b_HmiCmdStop := (#IOdi_HmiCmd.%X6 OR (#IOw_DCSCmd.%X4 AND #Ib_DCSPermissive)) OR #Ib_CmdGenDis;
	#b_HmiCmdRstAlm := #IOdi_HmiCmd.%X7;
	#IOdi_HmiCmd := 0;
	#IOw_DCSCmd := 0;


	// Mode change only possible if area is stopped
	IF #Ib_AreaStopped THEN
	    // Set Iu_CmdMode for ModeManager
	    #PML_ModeManager.Iu_CmdMode.Manual := #b_HmiCmdModMan;
	    #PML_ModeManager.Iu_CmdMode.Disabled := #b_HmiCmdModDis;
	    #PML_ModeManager.Iu_CmdMode.Production := #b_HmiCmdModAuto;

	    // If Mode command is given, mode change request = true
	    IF (#b_HmiCmdModMan OR #b_HmiCmdModDis OR #b_HmiCmdModAuto) THEN
	        #PML_ModeManager.IOb_CmdModeChangeRequest := TRUE;
	    ELSE
	        #PML_ModeManager.IOb_CmdModeChangeRequest := FALSE;
	    END_IF;

	END_IF;

	// Current state
	IF #b_StaRun THEN
	    #PML_ModeManager.Idi_StateCurrent := 6; // Execute State
	ELSE
	    #PML_ModeManager.Idi_StateCurrent := 2; // Stopped State
	END_IF;

	#PML_ModeManager();

	// If Cmd Simulation mode
	IF (#b_HmiCmdModSimOn) THEN
	    #b_StaSim := TRUE;
	ELSIF (#b_HmiCmdModSimOff) THEN
	    #b_StaSim := FALSE;
	END_IF;

	// If start and stop area
	IF (#b_HmiCmdStart) THEN
	    #b_StaRun := TRUE;
	END_IF;
	IF (#b_HmiCmdStop OR #Ib_CmdRstRelease OR #Ib_CmdGenMan) THEN
	    #b_StaRun := FALSE;
	END_IF;


	// Write outputs
	#Ob_StaExecute := #Ib_CmdGenRelease AND #b_StaRun;
	#Ob_StaAlm := #IOu_AreaFb.Alm.Alm;
	#Ob_StaWrn := #IOu_AreaFb.Alm.Wrn;
	#Ob_StaRstAlm := #Ib_CmdRstAlm OR #b_HmiCmdRstAlm;
	#Ob_StaSim := #b_StaSim;
	#b_StaAlm_Lvl1 := #IOu_AreaFb.Alm.Alm_Lvl1;
	#b_StaAlm_Lvl2 := #IOu_AreaFb.Alm.Alm_Lvl2;
	#b_StaAlm_Lvl3 := #IOu_AreaFb.Alm.Alm_Lvl3;

	// Area commands
	#Ou_AreaCmd.Alm.Rst := #Ib_CmdRstAlm OR #b_HmiCmdRstAlm;
	#Ou_AreaCmd.Mode.Man := #PML_ModeManager.Ou_ModeCurrent.Manual;
	#Ou_AreaCmd.Mode.Dis := #PML_ModeManager.Ou_ModeCurrent.Disabled;
	#Ou_AreaCmd.Mode.Auto := #PML_ModeManager.Ou_ModeCurrent.Production;
	#Ou_AreaCmd.Sim.ForceOff := #Ib_SimForceOff;
	#Ou_AreaCmd.Sim.ForceOn := #Ib_SimForceOn;
	#Ou_AreaCmd.Mode.AreaMode := #Ib_AreaCmdMode;

	// Write Current Mode UDT to output.
	#Ou_CurrentMode.Production := #PML_ModeManager.Ou_ModeCurrent.Production;
	#Ou_CurrentMode.Manual := #PML_ModeManager.Ou_ModeCurrent.Manual;
	#Ou_CurrentMode.Disabled := #PML_ModeManager.Ou_ModeCurrent.Disabled;

	// Status Area feedback
	#StaAreaFb.Alm.Alm := #IOu_AreaFb.Alm.Alm;
	#StaAreaFb.Alm.Wrn := #IOu_AreaFb.Alm.Wrn;
	#StaAreaFb.Alm.New := #IOu_AreaFb.Alm.New;
	#StaAreaFb.Alm.StopArea := #IOu_AreaFb.Alm.StopArea;

	// Reset Area feedback
	#IOu_AreaFb.Alm.Alm := FALSE;
	#IOu_AreaFb.Alm.Wrn := FALSE;
	#IOu_AreaFb.Alm.New := FALSE;
	#IOu_AreaFb.Alm.StopArea := FALSE;
	#IOu_AreaFb.Alm.Alm_Lvl1 := FALSE;
	#IOu_AreaFb.Alm.Alm_Lvl2 := FALSE;
	#IOu_AreaFb.Alm.Alm_Lvl3 := FALSE;


	// Copy state bits into double word for HMI
	#Odi_HmiSta.%X0 := #PML_ModeManager.Ou_ModeCurrent.Manual;
	#Odi_HmiSta.%X1 := #PML_ModeManager.Ou_ModeCurrent.Disabled;
	#Odi_HmiSta.%X2 := #PML_ModeManager.Ou_ModeCurrent.Production;
	#Odi_HmiSta.%X3 := #Ob_StaSim;
	#Odi_HmiSta.%X4 := #Ob_StaAlm;
	#Odi_HmiSta.%X5 := #Ob_StaWrn;
	#Odi_HmiSta.%X6 := #b_StaRun;
	#Odi_HmiSta.%X7 := #Ib_AreaStopped;
	#Odi_HmiSta.%X8 := #b_StaAlm_Lvl1;    //Animated Lvl1 area alarm status
	#Odi_HmiSta.%X9 := #b_StaAlm_Lvl2;    //Animated Lvl2 area alarm status
	#Odi_HmiSta.%X10 := #b_StaAlm_Lvl3;   //Animated Lvl3 area alarm status


	// Copy state bits into word for HMI
	#I_HmiSta.%X0 := #PML_ModeManager.Ou_ModeCurrent.Production;
	#I_HmiSta.%X1 := #PML_ModeManager.Ou_ModeCurrent.Manual;
	#I_HmiSta.%X2 := #PML_ModeManager.Ou_ModeCurrent.Disabled;
	#I_HmiSta.%X3 := #b_StaRun;
	#I_HmiSta.%X4 := NOT #b_StaRun;
	#I_HmiSta.%X7 := #Ib_AreaStopped;
	#I_HmiSta.%X8 := #Ob_StaAlm;
	#I_HmiSta.%X9 := #Ob_StaWrn;



END_FUNCTION_BLOCK

FUNCTION_BLOCK "FB_CM_AXV"
TITLE = Analog valve
{ S7_Optimized_Access := 'FALSE' }
AUTHOR : Reditech
FAMILY : Typical
VERSION : 0.0
//Reditech standard typical for controlling an analog valve
   VAR_INPUT
      Ib_FbPosOpn : Bool := FALSE;   //  feedback position open (failsafe : 0=open)
      Ib_FbPosCls : Bool := FALSE;   //  feedback position closed (failsafe : 0=closed)
      Ir_ActPos : Real;   //  Actual valve position (measurement)
      Ir_ParAutSp : Real;   //  automatic setpoint
      Ir_ParMaxPos : Real := 100.0;   //  Maximum position value
      Ir_ParMinPos : Real;   //  Minimum position value
      Ir_ParCtlDev : Real := 1.0;   //  Control deviation (for digital output and feedback OK)
      Ir_ParSafPos : Real;   //  Safety position
      Ir_ParMaxRaw : Real;   //  Max value for analogue output mode
      Ir_ParMinRaw : Real;   //  Min value for analogue output mode
      Ii_ParTO : Int := 5;   //  time out value for feedback monitoring
      Iby_Saf : Byte := 16#00;   //  8 safety bits : 1=error
      Iby_IlOn : Byte;   //  8 interlock bits : 1 prevents Pos1/opening
      Iby_IlOff { ExternalVisible := 'False'} : Byte;   //  8 interlock bits : 1 prevents Pos0/closing
      Ib_Pls1S : Bool;
      Ib_DisAlmWrn : Bool;
      Iw_Cfg : Word := 16#0000;   //  .0=analog pos present / .1=digital pos present
   END_VAR

   VAR_OUTPUT
      Or_SpOut : Real;   //  Control output
      Ow_SpRaw : Word;   //  Control output recalculated for analog output node
      Ob_Opn : Bool;   //  control output open
      Ob_Cls : Bool;   //  control output close
      Ob_PosOk : Bool;   //  Position reached
      Ob_Alm : Bool;   //  general alarm
      Ob_StaOpn : Bool;   //  Status in position 1
      Ob_StaCls : Bool;   //  Status in position 0
      Or_StaPos : Real;
      Odi_HmiSta : DInt;   //  State bits for HMI
      Oi_HmiAlm : Int;
      Odi_HmiAlm : DInt;   //  Alarm bit for HMI
   END_VAR

   VAR_IN_OUT
      IOr_ManSP : Real;   //  manual setpoint
      IOr_SimPos : Real := 0.0;   //  Simulated position
      IOdi_HmiCmd : DInt := 0;   //  Command bits from HMI
      IO_AreaCmd : "UDT_AreaCmd";   //  Command bits from area
      IO_AreaFb : "UDT_AreaFb";   //  Feedback bits to area
   END_VAR

   VAR
      i_TmrFbPos : Int;   //  timer feedback control
      b_HmiCmdModAut { ExternalAccessible := 'False'; ExternalVisible := 'False'; ExternalWritable := 'False'} : Bool;   //  command change mode to AUTO
      b_HmiCmdModMan { ExternalAccessible := 'False'; ExternalVisible := 'False'; ExternalWritable := 'False'} : Bool;   //  command change mode to MANUAL
      b_HmiCmdModDis { ExternalAccessible := 'False'; ExternalVisible := 'False'; ExternalWritable := 'False'} : Bool;   //  command change mode to DISABLED
      b_HmiCmdSim { ExternalAccessible := 'False'; ExternalVisible := 'False'; ExternalWritable := 'False'} : Bool;   //  toggle simulation mode
      b_HmiCmdRst { ExternalAccessible := 'False'; ExternalVisible := 'False'; ExternalWritable := 'False'} : Bool;   //  reset alarms
      b_StaModAut { ExternalAccessible := 'False'; ExternalVisible := 'False'; ExternalWritable := 'False'} : Bool;   //  state AUTOMATIC
      b_StaModMan { ExternalAccessible := 'False'; ExternalVisible := 'False'; ExternalWritable := 'False'} : Bool := TRUE;   //  state MANUAL
      b_StaModDis { ExternalAccessible := 'False'; ExternalVisible := 'False'; ExternalWritable := 'False'} : Bool;   //  state DISABLED
      b_StaSim { ExternalAccessible := 'False'; ExternalVisible := 'False'; ExternalWritable := 'False'} : Bool;   //  state simulation ON
      b_StaIlOff { ExternalAccessible := 'False'; ExternalVisible := 'False'; ExternalWritable := 'False'} : Bool;   //  state interlock OFF : 1 = interlocked (prevents closing)
      b_StaIlOn { ExternalAccessible := 'False'; ExternalVisible := 'False'; ExternalWritable := 'False'} : Bool;   //  state interlock ON : 1 = interlocked (prevents opening)
      b_StaSaf { ExternalAccessible := 'False'; ExternalVisible := 'False'; ExternalWritable := 'False'} : Bool;   //  state safety : 1 = error (valve to safety position)
      b_ReqOpn { ExternalAccessible := 'False'; ExternalVisible := 'False'; ExternalWritable := 'False'} : Bool;   //  output command open
      b_ReqCls { ExternalAccessible := 'False'; ExternalVisible := 'False'; ExternalWritable := 'False'} : Bool;   //  output command close
      b_StaPosOk { ExternalAccessible := 'False'; ExternalVisible := 'False'; ExternalWritable := 'False'} : Bool;   //  position (setpoint) reached
      b_StaAlm { ExternalAccessible := 'False'; ExternalVisible := 'False'; ExternalWritable := 'False'} : Bool;   //  general alarm
      b_CfgAnaPosPres { ExternalAccessible := 'False'; ExternalVisible := 'False'; ExternalWritable := 'False'} : Bool;   //  configuration : analog position feedback present
      b_CfgDigPosPres { ExternalAccessible := 'False'; ExternalVisible := 'False'; ExternalWritable := 'False'} : Bool;   //  configuration : digital limit positions present (min and max)
      b_CfgHldMod { ExternalAccessible := 'False'; ExternalVisible := 'False'; ExternalWritable := 'False'} : Bool;
      b_CfgDisableSim { ExternalAccessible := 'False'; ExternalVisible := 'False'; ExternalWritable := 'False'} : Bool;
      b_CfgStopArea { ExternalAccessible := 'False'; ExternalVisible := 'False'; ExternalWritable := 'False'} : Bool;
      b_AlmToFb { ExternalAccessible := 'False'; ExternalVisible := 'False'; ExternalWritable := 'False'} : Bool;   //  alarm time out feedback
      b_AlmFbInc { ExternalAccessible := 'False'; ExternalVisible := 'False'; ExternalWritable := 'False'} : Bool;   //  alarm inconsistent feedbacks (both together)
      b_AlmIncIl { ExternalAccessible := 'False'; ExternalVisible := 'False'; ExternalWritable := 'False'} : Bool;   //  alarm inconsistent interlocks (both together)
      b_ReqAut { ExternalAccessible := 'False'; ExternalVisible := 'False'; ExternalWritable := 'False'} : Bool;   //  automatic mode requested
      b_ReqMan { ExternalAccessible := 'False'; ExternalVisible := 'False'; ExternalWritable := 'False'} : Bool;   //  manual mode requested
      b_ReqDis { ExternalAccessible := 'False'; ExternalVisible := 'False'; ExternalWritable := 'False'} : Bool;   //  disabled mode requested
      b_TFbPos { ExternalAccessible := 'False'; ExternalVisible := 'False'; ExternalWritable := 'False'} : Bool;   //  tmer finished, feedback monitoring Pos1
      b_SpChange { ExternalAccessible := 'False'; ExternalVisible := 'False'; ExternalWritable := 'False'} : Bool;
      r_SpSel { ExternalAccessible := 'False'; ExternalVisible := 'False'; ExternalWritable := 'False'} : Real;   //  selected setpoint
      r_SpPrev { ExternalAccessible := 'False'; ExternalVisible := 'False'; ExternalWritable := 'False'} : Real;
      r_DevMax { ExternalAccessible := 'False'; ExternalVisible := 'False'; ExternalWritable := 'False'} : Real;
      r_DevMin { ExternalAccessible := 'False'; ExternalVisible := 'False'; ExternalWritable := 'False'} : Real;
      r_FrzVal { ExternalAccessible := 'False'; ExternalVisible := 'False'; ExternalWritable := 'False'} : Real;
      b_TStart : Bool;
      b_Tsim : Bool;
      FB_UTIL_TON_Instance_AXV_TEST : "FB_UTIL_TON_Sec";
      FB_UTIL_TON_Instance : "FB_UTIL_TON_Sec";
      i_TSim : Int;
      b_PrevTSim : Bool;
      r_ReqSP : Real;
      r_DevClsMaxEP : Real;
      r_DevClsMinEP : Real;
      r_DevOpnMaxEP : Real;
      r_DevOpnMinEP : Real;
      b_AlmIncInput : Bool;
      b_AlmOutOfBounds : Bool;
      b_AlmFbEP : Bool;
      b_CondOutOfBounds : Bool;
      b_DisAlmWrn : Bool;
      b_dummy : Bool;
      i_dummy : Int;
      b_StaAlmNew : Bool;
      b_NoAlm : Bool;
      i_AlmAck : Int;
      b_DisAlmWrn_1 : Bool;
      b_RstAlm : Bool;
      b_AutoMan_SP : Bool;   // HMI Selection for Automatic or Manual SetPoint 0->Man / 1->Auto
      I_HmiSta : Word;
      i_Category : Int := 1;   // Device alarm category setting
   END_VAR

   VAR_TEMP
      di_AUX : DInt;   //  auxiliary double word for calculation of state or alarm word to HMI
   END_VAR


BEGIN
	// =============================================================================================================================
	// Purpose: Reditech standard typical FOR controlling an analog valve
	// -----------------------------------------------------------------------------------------------------------------------------
	// Date (dd MMM yyyy) Developer                                   Version Comments/Reason FOR change
	// .................. .........                                   ....... ..........................
	// 18 Dec 2018        Bram Verheyen                               09.0    Full review
	// 30 Jan 2019        Matthias De Staelen                         09.1    Outputs can be high in simulation mode
	// =============================================================================================================================

	//============================================================================================
	#b_CfgAnaPosPres := #Iw_Cfg.%X0;
	#b_CfgDigPosPres := #Iw_Cfg.%X1;
	#b_CfgHldMod := #Iw_Cfg.%X2;
	#b_CfgDisableSim := #Iw_Cfg.%X10;
	#b_CfgStopArea := #Iw_Cfg.%X11;

	//============================================================================================
	#b_DisAlmWrn := #Ib_DisAlmWrn OR #IO_AreaCmd.Alm.Dis OR #b_StaModDis;

	//============================================================================================
	#b_StaSaf := (#Iby_Saf <> 0);
	#b_StaIlOn := (#Iby_IlOn <> 0);
	#b_StaIlOff := (#Iby_IlOff <> 0);

	//============================================================================================
	#b_HmiCmdModAut := #IOdi_HmiCmd.%X0;
	#b_HmiCmdModMan := #IOdi_HmiCmd.%X1;
	#b_HmiCmdModDis := #IOdi_HmiCmd.%X2;
	#b_HmiCmdSim := #IOdi_HmiCmd.%X3;
	#b_HmiCmdRst := #IOdi_HmiCmd.%X4;
	#IOdi_HmiCmd := 0;

	//============================================================================================
	IF #IO_AreaCmd.Mode.AreaMode THEN
	    #b_ReqAut := #IO_AreaCmd.Mode.Auto;
	    #b_ReqMan := #IO_AreaCmd.Mode.Man;
	    #b_ReqDis := #IO_AreaCmd.Mode.Dis;
	ELSE
	    IF #b_CfgHldMod THEN
	        #b_ReqAut := #b_HmiCmdModAut;
	        #b_ReqMan := #b_HmiCmdModMan;
	        #b_ReqDis := #b_HmiCmdModDis;
	    ELSE
	        #b_ReqAut := #b_HmiCmdModAut AND NOT #b_StaAlm AND NOT #b_StaSaf;
	        #b_ReqMan := #b_HmiCmdModMan OR ((#b_StaAlm OR #b_StaSaf) AND NOT #b_StaModDis);
	        #b_ReqDis := #b_HmiCmdModDis;
	    END_IF;
	END_IF;
	IF (#b_ReqAut AND NOT #b_ReqMan AND NOT #b_ReqDis) THEN
	    #b_StaModAut := true;
	    #b_StaModMan := false;
	    #b_StaModDis := false;
	END_IF;
	IF (#b_ReqMan AND NOT #b_ReqAut AND NOT #b_ReqDis) THEN
	    #b_StaModAut := false;
	    #b_StaModMan := true;
	    #b_StaModDis := false;
	END_IF;
	IF (#b_ReqDis AND NOT #b_ReqMan AND NOT #b_ReqAut) THEN
	    #b_StaModAut := false;
	    #b_StaModMan := false;
	    #b_StaModDis := true;
	END_IF;

	//============================================================================================
	IF #IO_AreaCmd.Sim.ForceOn OR (#b_HmiCmdSim AND NOT #b_StaSim AND NOT #IO_AreaCmd.Sim.ForceOn AND NOT #IO_AreaCmd.Sim.ForceOff) THEN
	    #b_StaSim := true;
	    #b_HmiCmdSim := false; // reset of command necessary, else simulation will always be reset immediately by following instructions
	END_IF;
	IF #IO_AreaCmd.Sim.ForceOff OR (#b_HmiCmdSim AND #b_StaSim AND NOT #IO_AreaCmd.Sim.ForceOn AND NOT #IO_AreaCmd.Sim.ForceOff) THEN
	    #b_StaSim := false;
	    #b_HmiCmdSim := false;
	END_IF;

	//============================================================================================
	// automatic feedback simulation
	#r_DevMax := #r_SpSel + #Ir_ParCtlDev;
	#r_DevMin := #r_SpSel - #Ir_ParCtlDev;
	IF #b_StaSim AND "Clock_10Hz" THEN
	    IF (#IOr_SimPos <= #r_DevMin) THEN
	        #IOr_SimPos := #IOr_SimPos + #Ir_ParCtlDev;
	    END_IF;
	    IF (#IOr_SimPos >= #r_DevMax) THEN
	        #IOr_SimPos := #IOr_SimPos - #Ir_ParCtlDev;
	    END_IF;
	END_IF;

	// Select valve position
	IF #b_StaSim THEN
	    #Or_StaPos := #IOr_SimPos;
	END_IF;
	IF NOT #b_StaSim AND #b_CfgAnaPosPres THEN
	    #Or_StaPos := #Ir_ActPos;
	END_IF;
	IF NOT #b_StaSim AND NOT #b_CfgAnaPosPres AND #b_CfgDigPosPres AND #Ob_StaOpn THEN
	    #Or_StaPos := #Ir_ParMaxPos;
	END_IF;
	IF NOT #b_StaSim AND NOT #b_CfgAnaPosPres AND #b_CfgDigPosPres AND #Ob_StaCls THEN
	    #Or_StaPos := #Ir_ParMinPos;
	END_IF;
	IF NOT #b_StaSim AND NOT #b_CfgAnaPosPres AND NOT #b_CfgDigPosPres THEN
	    #Or_StaPos := #Or_SpOut;
	END_IF;

	//============================================================================================
	// Digital feedback, selection simulation or real time
	#Ob_StaOpn := (NOT #b_StaSim AND (#b_CfgDigPosPres AND #Ib_FbPosOpn))
	OR (NOT #b_StaSim AND (NOT #b_CfgDigPosPres AND (#Or_StaPos >= #r_DevOpnMinEP)))
	OR (#b_StaSim AND (#Or_StaPos > #r_DevClsMaxEP));

	#Ob_StaCls := (NOT #b_StaSim AND (#b_CfgDigPosPres AND #Ib_FbPosCls))
	OR (NOT #b_StaSim AND (NOT #b_CfgDigPosPres AND (#Or_StaPos <= #r_DevClsMaxEP)))
	OR (#b_StaSim AND (#Or_StaPos <= #r_DevClsMaxEP));

	// If the valve position is between 1% and 100%, shows color purple
	IF (#Or_StaPos > 1.0) AND (#Or_StaPos < 100.0)
	THEN
	    #Odi_HmiSta.%X8 := TRUE;
	ELSE
	    #Odi_HmiSta.%X8 := FALSE;
	END_IF;

	// Setpoint feedback check
	#b_StaPosOk := (NOT #b_CfgAnaPosPres) OR
	(#b_CfgAnaPosPres AND (#Ir_ActPos >= (#Or_SpOut - #Ir_ParCtlDev)) AND (#Ir_ActPos <= (#Or_SpOut + #Ir_ParCtlDev)));
	#Ob_PosOk := #b_StaPosOk AND NOT #b_StaAlm;

	//============================================================================================
	#b_SpChange := (#r_SpSel <> #r_SpPrev);
	#r_SpPrev := #r_SpSel;

	//============================================================================================
	(*lower and higher deviation values from the endpoint*)
	#r_DevClsMaxEP := #Ir_ParMinPos + #Ir_ParCtlDev;
	#r_DevClsMinEP := #Ir_ParMinPos - #Ir_ParCtlDev;
	#r_DevOpnMaxEP := #Ir_ParMaxPos + #Ir_ParCtlDev;
	#r_DevOpnMinEP := #Ir_ParMaxPos - #Ir_ParCtlDev;

	//============================================================================================
	#b_NoAlm := false;
	#b_RstAlm := #b_HmiCmdRst OR #IO_AreaCmd.Alm.Rst;
	"FC_UTIL_AlmAck"(Ib_CmdAck := #b_RstAlm,
	                 Oi_StaAlm => #i_dummy,
	                 Ob_StaAlm => #b_dummy,
	                 Ob_StaNewAlm => #b_StaAlmNew,
	                 IO_Alm0 := #b_AlmToFb,
	                 IO_Alm1 := #b_AlmFbInc,
	                 IO_Alm2 := #b_AlmIncIl,
	                 IO_Alm3 := #b_AlmOutOfBounds,
	                 IO_Alm4 := #b_AlmFbEP,
	                 IO_Alm5 := #b_AlmIncInput,
	                 IO_Alm6 := #b_NoAlm,
	                 IO_Alm7 := #b_NoAlm,
	                 IO_Alm8 := #b_NoAlm,
	                 IO_Alm9 := #b_NoAlm,
	                 IO_Alm10 := #b_NoAlm,
	                 IO_Alm11 := #b_NoAlm,
	                 IO_Alm12 := #b_NoAlm,
	                 IO_Alm13 := #b_NoAlm,
	                 IO_Alm14 := #b_NoAlm,
	                 IO_Alm15 := #b_NoAlm,
	                 IOi_StaAck := #i_AlmAck);


	//============================================================================================
	IF #Ii_ParTO > 0 THEN  // only when time value > 0
	    #FB_UTIL_TON_Instance_AXV_TEST(Ib_In := (#b_CfgAnaPosPres AND NOT #b_StaPosOk AND NOT #b_SpChange AND NOT #b_StaSim),
	                                   Ii_Base := 1,
	                                   Ib_Hold := 0,
	                                   Ii_tValue := #Ii_ParTO,
	                                   Oi_tmrValue => #i_TmrFbPos,
	                                   Ob_Out => #b_TFbPos);
	END_IF;

	IF (#b_TFbPos AND (#Ii_ParTO > 0))
	    AND NOT #b_DisAlmWrn THEN
	    #b_AlmToFb := true;
	END_IF;

	//============================================================================================
	IF (#r_ReqSP > #Ir_ParMaxPos
	    OR #r_ReqSP < #Ir_ParMinPos
	    OR (#Ir_ParSafPos > 0 AND (#Ir_ParSafPos > #Ir_ParMaxPos OR #Ir_ParSafPos < #Ir_ParMinPos)))
	    AND NOT #b_DisAlmWrn THEN
	    #b_AlmOutOfBounds := true;
	END_IF;

	//============================================================================================
	IF ((#Ir_ActPos > #r_DevOpnMaxEP OR #Ir_ActPos < #r_DevClsMinEP) AND #b_CfgAnaPosPres)
	    AND NOT #b_DisAlmWrn THEN
	    #b_AlmIncInput := 1;
	END_IF;

	//============================================================================================
	IF (#Ob_StaOpn AND #Ob_StaCls)
	    AND NOT #b_DisAlmWrn THEN
	    #b_AlmFbInc := 1;
	END_IF;

	//============================================================================================
	IF (#b_CfgAnaPosPres
	    AND #b_CfgDigPosPres
	    AND ((#Ib_FbPosCls AND #Ir_ActPos > #r_DevClsMaxEP) OR (#Ib_FbPosOpn AND #Ir_ActPos < #r_DevOpnMinEP)))
	    AND NOT #b_DisAlmWrn THEN
	    #b_AlmFbEP := true;
	END_IF;

	//============================================================================================
	IF (#b_StaIlOn AND #b_StaIlOff) AND NOT #b_DisAlmWrn THEN
	    #b_AlmIncIl := true;
	END_IF;
	IF NOT (#b_StaIlOn AND #b_StaIlOff) THEN
	    #b_AlmIncIl := false;
	END_IF;

	//============================================================================================
	#b_StaAlm := #b_AlmOutOfBounds OR #b_AlmToFb OR #b_StaSaf OR #b_AlmFbInc OR #b_AlmIncIl OR #b_AlmIncInput OR #b_AlmFbEP OR (#Iby_IlOn>0) OR (#Iby_IlOff>0);
	#Ob_Alm := #b_StaAlm;

	//============================================================================================
	IF #b_StaModAut THEN
	    #r_ReqSP := #Ir_ParAutSp;
	END_IF;

	//============================================================================================
	IF #b_StaModMan THEN
	    #r_ReqSP := #IOr_ManSP;
	END_IF;

	//============================================================================================
	IF #b_StaModAut OR #b_StaModMan THEN
	    (*go to min pos*)
	    IF (#b_StaIlOn AND #b_CfgAnaPosPres) THEN
	        #r_SpSel := #Ir_ParMinPos;
	        #IOr_ManSP := #Ir_ParMinPos;

	        (*hold condition*)
	    ELSIF (#b_StaIlOff AND #b_CfgAnaPosPres) THEN
	        #r_SpSel := #r_FrzVal;
	        #IOr_ManSP := #r_FrzVal;

	        (*follows setpoint as usual*)
	    ELSE
	        #r_SpSel := #r_ReqSP;
	    END_IF;
	END_IF;

	IF (#b_StaSaf OR #b_StaAlm) THEN
	    IF #Ir_ParSafPos > 0 THEN
	        #r_SpSel := #Ir_ParSafPos;
	    ELSE
	        #r_SpSel := #r_FrzVal;
	    END_IF;
	ELSIF (#b_AlmToFb OR #b_AlmIncInput) THEN
	    #r_SpSel := #r_FrzVal;
	END_IF;

	IF #b_StaIlOn THEN
	    #r_SpSel := #Ir_ParMinPos;
	END_IF;

	IF #b_StaModDis THEN
	    #r_SpSel := 0.0;
	    #IOr_ManSP := 0.0;
	END_IF;

	//============================================================================================
	#b_ReqOpn := (#Or_StaPos < #r_DevMin) AND NOT #b_StaAlm AND NOT #b_StaIlOn AND NOT #b_StaModDis AND NOT #Ob_StaOpn;
	#b_ReqCls := (#Or_StaPos > #r_DevMax) AND NOT #b_StaAlm AND NOT #b_StaIlOff AND NOT #b_StaModDis AND NOT #Ob_StaCls;

	//============================================================================================
	// Output position
	#Or_SpOut := #r_SpSel;
	#Ob_Opn := #b_ReqOpn;
	#Ob_Cls := #b_ReqCls;

	// recalculate output to word value for analog output node
	IF ((#Ir_ParMaxPos - #Ir_ParMinPos) > 0.0) THEN  // check if division by positive number
	    #Ow_SpRaw := INT_TO_WORD(IN := (REAL_TO_INT(IN := ((((#r_SpSel - #Ir_ParMinPos) / (#Ir_ParMaxPos - #Ir_ParMinPos)) * (#Ir_ParMaxRaw - #Ir_ParMinRaw)) + #Ir_ParMinRaw))));
	ELSE
	    #Ow_SpRaw := 0;
	END_IF;

	//============================================================================================
	IF NOT #b_AlmToFb
	    AND NOT #b_AlmFbInc
	    AND NOT #b_AlmIncIl
	    AND NOT #b_AlmOutOfBounds
	    AND NOT #b_AlmFbEP
	    AND NOT #b_AlmIncInput
	    AND NOT #b_StaIlOff THEN
	    #r_FrzVal := #Ir_ActPos;
	END_IF;

	//============================================================================================
	#Odi_HmiSta.%X0 := #b_StaModAut;
	#Odi_HmiSta.%X1 := #b_StaModMan;
	#Odi_HmiSta.%X2 := #b_StaModDis;
	#Odi_HmiSta.%X3 := #b_StaSim;
	#Odi_HmiSta.%X4 := #b_StaIlOff;
	#Odi_HmiSta.%X5 := #b_StaIlOn;
	#Odi_HmiSta.%X6 := #b_StaSaf;
	#Odi_HmiSta.%X7 := #b_StaSim;
	#Odi_HmiSta.%X16 := #b_ReqOpn;
	#Odi_HmiSta.%X17 := #b_ReqCls;
	#Odi_HmiSta.%X18 := #b_StaPosOk;
	#Odi_HmiSta.%X19 := #Ob_StaOpn;
	#Odi_HmiSta.%X20 := #Ob_StaCls;
	#Odi_HmiSta.%X21 := #b_StaAlm;
	#Odi_HmiSta.%X24 := #b_CfgAnaPosPres;
	#Odi_HmiSta.%X25 := #b_CfgDigPosPres;
	#Odi_HmiSta.%X26 := #b_CfgHldMod;
	#Odi_HmiSta.%X28 := #IO_AreaCmd.Mode.AreaMode;

	#I_HmiSta.%X0 := #b_StaModAut;
	#I_HmiSta.%X1 := #b_StaModMan;
	#I_HmiSta.%X2 := #b_StaModDis;
	#I_HmiSta.%X3 := #b_StaSim;

	IF #Or_StaPos = 100.0 THEN
	    #I_HmiSta.%X4 := TRUE;
	ELSE
	    #I_HmiSta.%X4 := FALSE;
	END_IF;

	#I_HmiSta.%X5 := #Ob_StaCls;
	#I_HmiSta.%X6 := #Odi_HmiSta.%X8; //Between 0% and 100%
	#I_HmiSta.%X7 := #b_StaAlm;

	//============================================================================================
	#di_AUX := 0;
	#di_AUX.%X0 := #b_AlmToFb;
	#di_AUX.%X1 := #b_AlmFbInc;
	#di_AUX.%X2 := #b_AlmIncIl;
	#di_AUX.%X3 := #b_AlmOutOfBounds;
	#di_AUX.%X4 := #b_AlmFbEP;
	#di_AUX.%X5 := #b_AlmIncInput;
	#di_AUX.%X8 := #Iby_IlOff.%X0;
	#di_AUX.%X9 := #Iby_IlOff.%X1;
	#di_AUX.%X10 := #Iby_IlOff.%X2;
	#di_AUX.%X11 := #Iby_IlOff.%X3;
	#di_AUX.%X12 := #Iby_IlOff.%X4;
	#di_AUX.%X13 := #Iby_IlOff.%X5;
	#di_AUX.%X14 := #Iby_IlOff.%X6;
	#di_AUX.%X15 := #Iby_IlOff.%X7;
	#di_AUX.%X16 := #Iby_IlOn.%X0;
	#di_AUX.%X17 := #Iby_IlOn.%X1;
	#di_AUX.%X18 := #Iby_IlOn.%X2;
	#di_AUX.%X19 := #Iby_IlOn.%X3;
	#di_AUX.%X20 := #Iby_IlOn.%X4;
	#di_AUX.%X21 := #Iby_IlOn.%X5;
	#di_AUX.%X22 := #Iby_IlOn.%X6;
	#di_AUX.%X23 := #Iby_IlOn.%X7;
	#di_AUX.%X24 := #Iby_Saf.%X0;
	#di_AUX.%X25 := #Iby_Saf.%X1;
	#di_AUX.%X26 := #Iby_Saf.%X2;
	#di_AUX.%X27 := #Iby_Saf.%X3;
	#di_AUX.%X28 := #Iby_Saf.%X4;
	#di_AUX.%X29 := #Iby_Saf.%X5;
	#di_AUX.%X30 := #Iby_Saf.%X6;
	#di_AUX.%X31 := #Iby_Saf.%X7;
	#Odi_HmiAlm := #di_AUX;

	//============================================================================================
	#di_AUX := 0;
	#di_AUX.%X0 := #b_AlmToFb;
	#di_AUX.%X1 := #b_AlmFbInc;
	#di_AUX.%X2 := #b_AlmIncIl;
	#di_AUX.%X3 := #b_AlmOutOfBounds;
	#di_AUX.%X4 := #b_AlmFbEP;
	#di_AUX.%X5 := #b_AlmIncInput;
	#Oi_HmiAlm := DINT_TO_INT(#di_AUX);

	//============================================================================================
	IF #b_StaModDis THEN
	    #IO_AreaFb.Mode.Dis := TRUE;
	END_IF;
	IF #b_StaModMan THEN
	    #IO_AreaFb.Mode.Man := TRUE;
	END_IF;
	IF #b_StaModAut THEN
	    #IO_AreaFb.Mode.Auto := TRUE;
	END_IF;
	IF #b_StaAlm THEN
	    #IO_AreaFb.Alm.Alm := TRUE;
	END_IF;
	IF #b_StaAlmNew THEN
	    #IO_AreaFb.Alm.New := TRUE;
	END_IF;
	IF #b_StaSim THEN
	    #IO_AreaFb.Sim.Sim := TRUE;
	END_IF;
	IF #b_StaAlm AND #b_CfgStopArea THEN
	    #IO_AreaFb.Alm.StopArea := TRUE;
	END_IF;

	//Generating alarm category feedback
	IF #i_Category = 1 AND #b_StaAlm THEN
	    #IO_AreaFb.Alm.Alm_Lvl1 := TRUE;
	END_IF;

	IF #i_Category = 2 AND #b_StaAlm THEN
	    #IO_AreaFb.Alm.Alm_Lvl2 := TRUE;
	END_IF;

	IF #i_Category = 3 AND #b_StaAlm THEN
	    #IO_AreaFb.Alm.Alm_Lvl3 := TRUE;
	END_IF;
END_FUNCTION_BLOCK


FUNCTION_BLOCK "FB_EM_Lvl_3Eqp"
{ S7_Optimized_Access := 'FALSE' }
VERSION : 0.1
   VAR_INPUT
      Ib_RequestEqp { ExternalVisible := 'False'} : Bool;   //  Request equipment Command
      Ib_LvlOff_FirstEqp : Bool;   //  Level switch low low
      Ib_LvlOff_SecondEqp : Bool;   //  Level switch low
      Ib_LvlOff_ThirdEqp : Bool;
      Ib_LvlOn_FirstEqp : Bool;   //  Level switch high
      Ib_LvlOn_SecondEqp : Bool;   //  Level switch High High
      Ib_LvlOn_ThirdEqp : Bool;
      Ib_NrEqp : Int;   //  Number of equipment used at the same time, 0 = 1 eqp, 1 = 2 eqp
   END_VAR

   VAR_OUTPUT
      Ob_ReqFirstEqp : Bool;   //  Request first equipment
      Ob_ReqSecondEqp : Bool;   //  Request second equipment
      Ob_ReqThirdEqp : Bool;
   END_VAR

   VAR_IN_OUT
      IO_AreaCmd : "UDT_AreaCmd";   //  Command bits from area
      IO_AreaFb : "UDT_AreaFb";   //  Feedback bits to area
   END_VAR

   VAR
      b_FirstEqpReq : Bool;   //  Request to Equipment 1
      b_SecondEqpReq : Bool;   //  Request to Equipment 2
      b_ThirdEqpReq : Bool;
      b_ReqAut : Bool;   //  Request automatic mode
      b_ReqMan : Bool;
      b_ReqDis : Bool;
   END_VAR


BEGIN
	//not used// =========================================================================================================================
	// Purpose: Reditech standard typical for controlling Pump Toggle manual automatic or semi-automatic
	// -------------------------------------------------------------------------------------------------------------------------
	// Date (dd MMM yyyy)   Developer                                   Version Comments/Reason for change
	// ..................   .........                                   ....... ..........................
	// 16 OCT 2018          Robin Cardinaels                               01      Initial (creation)
	// 31 JUL 2020          Ivan Galhardoni                                02      Implemented third Eqp for control
	// =========================================================================================================================
	// copy command bits from HMI and reset

	#b_ReqAut := #IO_AreaCmd.Mode.Auto;
	#b_ReqMan := #IO_AreaCmd.Mode.Man;
	#b_ReqDis := #IO_AreaCmd.Mode.Dis;

	IF NOT #b_ReqAut THEN
	    #b_FirstEqpReq := #b_SecondEqpReq := #b_ThirdEqpReq := false;
	ELSE
	    IF #Ib_LvlOn_FirstEqp THEN
	        #b_FirstEqpReq := TRUE;
	    END_IF;
	    IF #Ib_LvlOff_FirstEqp THEN
	        #b_FirstEqpReq := FALSE;
	    END_IF;

	    IF #Ib_NrEqp >= 2 THEN
	        // setting control bits for anaog and digital control.
	        IF #Ib_LvlOn_SecondEqp THEN
	            #b_SecondEqpReq := TRUE;
	        END_IF;
	        IF #Ib_LvlOff_SecondEqp THEN
	            #b_SecondEqpReq := FALSE;
	        END_IF;
	    ELSE
	        #b_SecondEqpReq := false;
	    END_IF;

	    IF #Ib_NrEqp = 3 THEN
	        // setting control bits for anaog and digital control.
	        IF #Ib_LvlOn_ThirdEqp THEN
	            #b_ThirdEqpReq := TRUE;
	        END_IF;
	        IF #Ib_LvlOff_ThirdEqp THEN
	            #b_ThirdEqpReq := FALSE;
	        END_IF;
	    ELSE
	        #b_ThirdEqpReq := false;
	    END_IF;

	END_IF;

	// Set Output For Motor 1
	#Ob_ReqFirstEqp := #Ib_RequestEqp AND #b_FirstEqpReq;

	//Set output for Motor 2
	#Ob_ReqSecondEqp := #Ib_RequestEqp AND #b_SecondEqpReq;

	//Set output for Motor 3
	#Ob_ReqThirdEqp := #Ib_RequestEqp AND #b_ThirdEqpReq;

END_FUNCTION_BLOCK

FUNCTION_BLOCK "FB_CM_Machine_Status"
{ S7_Optimized_Access := 'FALSE' }
VERSION : 0.1
   VAR_INPUT
      Ib_RunReq : Bool;   // Request to Start Disk Filter
      Ib_Sta_Run : Bool;   // Feedback from DiskFilter of Running Mode
      Ib_Sta_Fail : Bool;   // Feedback from DiskFilter of Failure Mode
      Iby_IlFwd { ExternalVisible := 'False'} : Byte;   //  8 interlock bits : 1 prevents run forward
      Ib_Ext_Signal : Bool;   // External signal dedicated for general purpouse action
      Ib_DisAlmWrn : Bool;   // Command to Disable Alarm
      Ib_ErrorEqp1 : Bool;   // Eqp 1 error or fault
      Ib_ErrorEqp2 : Bool;   // Eqp 2 error or fault
      Ib_StaEqp1 : Bool;   // Eqp 1 feedback stand alone
      Ib_StaEqp2 : Bool;   // Eqp 2 feedback stand alone
   END_VAR

   VAR_OUTPUT
      Ob_StartReq : Bool;   // Request to Disk Filter go to Running mode
      Ob_StaAlm : Bool;   // Feedback Alarm
      Odi_HmiSta : DInt;   //  State bits for HMI
      Oi_HmiAlm : Int;   //  Alarm bit for HMI
      Odi_ActCouRst : DInt := 0;   //  Actuation counter from last reset
      Odi_ActCouTot : DInt := 0;   //  Total actuation counter
      Odi_RunTimRst : DInt;   //  Operating hours from last reset
      Odi_RunTimTot : DInt;   //  Total operating hours
      Ob_StaRunning : Bool;   // Inform that the equipment is ready to operate
   END_VAR

   VAR_IN_OUT
      IO_AreaCmd : "UDT_AreaCmd";   //  Command bits from area
      IOdi_HmiCmd : DInt;   //  Command bits from HMI
      IO_AreaFb : "UDT_AreaFb";   //  Feedback bits to area
      Ii_ParTFb : Int := 5;   //  time out value for feedback monitoring
   END_VAR

   VAR
      b_RunReq : Bool;
      b_Running : Bool;
      b_Failure : Bool;
      b_General_Purpouse : Bool;
      b_NoAlm : Bool;
      b_RstAlm : Bool;
      b_dummy : Bool;
      i_dummy : Int;
      i_AlmAck : Int;
      b_StaAlmNew : Bool;
      b_CmdAutoStart : Bool;
      b_CmdReqStart : Bool;   // Commando to Request to Start System
      b_CmdStart : Bool;   // Commando to Start System
      b_ReqAut { ExternalVisible := 'False'} : Bool;   //  automatic mode requested
      b_ReqMan { ExternalVisible := 'False'} : Bool;   //  manual mode requested
      b_ReqDis { ExternalVisible := 'False'} : Bool;   //  disabled mode requested
      b_DisAlmWrn : Bool;
      b_StatusReady : Bool;
      FB_UTIL_Work_H_Rst : "FB_UTIL_Work_H";
      FB_UTIL_Work_H_Tot : "FB_UTIL_Work_H";
      FB_UTIL_TON_Del_1 { ExternalVisible := 'False'} : "FB_UTIL_TON_Sec";
      b_FbErrRun { S7_SetPoint := 'True'} : Bool;   // Error to go to Run Mode Feedback
      b_StaSim { ExternalVisible := 'False'} : Bool;   //  state simulation ON
      b_HmiCmdModAut { ExternalVisible := 'False'} : Bool;   //  command change mode to AUTO
      b_HmiCmdModMan { ExternalVisible := 'False'} : Bool;   //  command change mode to MANUAL
      b_HmiCmdModDis { ExternalVisible := 'False'} : Bool;   //  command change mode to DISABLED
      b_HmiCmdSim { ExternalVisible := 'False'} : Bool;   //  toggle simulation mode
      b_HmiCmdStartReq { ExternalVisible := 'False'} : Bool;   //  command Start
      b_HmiCmdStp { ExternalVisible := 'False'} : Bool;   //  command stop
      b_HmiCmdRst { ExternalVisible := 'False'} : Bool;   //  reset alarms
      b_HmiCmdRstActOpe { ExternalVisible := 'False'} : Bool;   //  reset actuation counter and operating hours
      b_StaModAut { ExternalVisible := 'False'} : Bool;   //  state AUTOMATIC
      b_StaModMan { ExternalVisible := 'False'} : Bool := TRUE;   //  state MANUAL
      b_StaModDis { ExternalVisible := 'False'} : Bool;   //  state DISABLED
      b_StaAlm { ExternalVisible := 'False'} : Bool;   //  general alarm
      b_FbSimStart { ExternalVisible := 'False'} : Bool;   //  internal feedback simulation
      b_Old_Ob_Run : Bool;
      b_StaIlOn { ExternalVisible := 'False'} : Bool;   //  state interlock ON : 1 = interlocked (prevents forward)
      b_AlmtoFb : Bool;
   END_VAR

   VAR_TEMP
      di_AUX : Int;   //  auxiliary double word for calculation of state or alarm word to HMI
   END_VAR


BEGIN
	// =============================================================================================================================
	// Purpose: Reditech standard typical to Communicate with any Field Machine
	// -----------------------------------------------------------------------------------------------------------------------------
	// Date (dd MMM yyyy)   Developer                   Version Comments/Reason for change
	// ..................   .........                   ....... ..........................
	// 22 May 2020          Willian Barroso               0.10    First Issue
	// 22 Jun 2020          Willian Barroso               0.20    Add Interlock Input
	// 09 Jul 2020          Ivan Galhardoni               1.00    Performed several changes in the simulation mode,HMI communication data and Auto/Man control
	// 08 Jul 2021          Ivan Galhardoni               1.01    Was changed the output command to a set command
	// =============================================================================================================================

	// =============================================================================================================================
	// Read Input Signals
	#b_RunReq := #Ib_RunReq;
	#b_Running := #Ib_Sta_Run;
	#b_General_Purpouse := #Ib_Ext_Signal;

	// =============================================================================================================================
	// Alarm Disable
	#b_DisAlmWrn := #Ib_DisAlmWrn OR #IO_AreaCmd.Alm.Dis OR #b_StaModDis;

	// =============================================================================================================================
	#b_StaIlOn := (#Iby_IlFwd <> 0);

	// =============================================================================================================================
	// HMI Commands
	//#b_HmiCmdModAut := #IOdi_HmiCmd.%X0;
	//#b_HmiCmdModMan := #IOdi_HmiCmd.%X1;
	//#b_HmiCmdModDis := #IOdi_HmiCmd.%X2;
	#b_HmiCmdSim := #IOdi_HmiCmd.%X3;       //Command to request simulation mode
	#b_HmiCmdStp := #IOdi_HmiCmd.%X4;       //Command to request machine to stop
	#b_HmiCmdRst := #IOdi_HmiCmd.%X5;       //Machine faceplate alarm reset command
	#b_HmiCmdStartReq := #IOdi_HmiCmd.%X6;  //Command to request machine start-up
	#b_HmiCmdRstActOpe := #IOdi_HmiCmd.%X8; //Number of starts reset button
	#IOdi_HmiCmd := 0;  //Erasing HMI commands
	// =============================================================================================================================
	// Area Mode
	IF #IO_AreaCmd.Mode.AreaMode THEN
	    #b_ReqAut := #IO_AreaCmd.Mode.Auto;
	    #b_ReqMan := #IO_AreaCmd.Mode.Man;
	    #b_ReqDis := #IO_AreaCmd.Mode.Dis;
	END_IF;

	IF (#b_ReqAut AND NOT #b_ReqMan AND NOT #b_ReqDis) THEN
	    #b_StaModAut := true;
	    #b_StaModMan := false;
	    #b_StaModDis := false;
	END_IF;
	IF (#b_ReqMan AND NOT #b_ReqAut AND NOT #b_ReqDis) THEN
	    #b_StaModAut := false;
	    #b_StaModMan := true;
	    #b_StaModDis := false;
	END_IF;
	IF (#b_ReqDis AND NOT #b_ReqAut AND NOT #b_ReqMan) THEN
	    #b_StaModAut := false;
	    #b_StaModMan := false;
	    #b_StaModDis := true;
	END_IF;

	// =============================================================================================================================
	// Simulation Mode
	IF #IO_AreaCmd.Sim.ForceOn OR (#b_HmiCmdSim AND NOT #b_StaSim AND NOT #IO_AreaCmd.Sim.ForceOn AND NOT #IO_AreaCmd.Sim.ForceOff) THEN
	    #b_StaSim := true;
	    #b_HmiCmdSim := false; // reset of command necessary, else simulation will always be reset immediately by following instructions
	END_IF;
	IF #IO_AreaCmd.Sim.ForceOff OR (#b_HmiCmdSim AND #b_StaSim AND NOT #IO_AreaCmd.Sim.ForceOn AND NOT #IO_AreaCmd.Sim.ForceOff) THEN
	    #b_StaSim := false;
	    #b_HmiCmdSim := false;
	END_IF;

	// =============================================================================================================================
	// Start Command Request
	IF (#b_RunReq AND NOT #b_CmdAutoStart AND NOT #b_StaModMan) OR (#b_StaModAut AND #b_RunReq AND #b_StaSim) OR #b_HmiCmdStartReq THEN //Command being requested by block input or HMI button
	    #b_CmdAutoStart := TRUE;
	END_IF;

	IF (#b_StaModAut AND #b_CmdAutoStart) OR (#b_StaModMan AND #b_CmdAutoStart) THEN
	    #b_CmdStart := TRUE;
	END_IF;

	IF (#b_CmdStart AND NOT #b_StaAlm AND NOT #b_StaModDis AND NOT #b_StaIlOn) THEN
	    #b_CmdReqStart := TRUE; //Final logic for start command request
	END_IF;

	//If There is a fault, or Hmi button request to stop, set command off
	IF #b_StaAlm OR #b_StaIlOn OR #b_StaModDis
	    OR (#b_StaModMan AND  #b_HmiCmdStp)
	    OR (#b_StaModAut AND NOT #b_RunReq) THEN
	    #b_CmdReqStart := FALSE;
	    #b_CmdStart := FALSE;
	    #b_CmdAutoStart := FALSE;
	    #b_FbSimStart := FALSE;
	END_IF;
	// =============================================================================================================================
	// Simulation of Start Command Request
	IF #b_StaSim THEN //Avoiding equipment start-up in simulation mode
	    #Ob_StartReq := FALSE;
	ELSE
	    #Ob_StartReq := #b_CmdReqStart;
	END_IF;

	// =============================================================================================================================
	// reset simulated feedback when starting to move
	IF NOT #b_StaSim OR #b_HmiCmdStp OR #b_StaAlm THEN
	    #b_FbSimStart := false;
	END_IF;

	// set simulated feedback
	IF #b_CmdReqStart AND #b_StaSim THEN
	    #b_FbSimStart := true;
	END_IF;

	// =============================================================================================================================
	// feedback, selection simulation or real time
	#Ob_StaRunning := (NOT #b_StaSim AND #b_Running) OR (#b_StaSim AND #b_FbSimStart);

	// =============================================================================================================================
	//Alarm Acknowledge
	#b_NoAlm := false;
	#b_RstAlm := #b_HmiCmdRst OR #IO_AreaCmd.Alm.Rst;
	"FC_UTIL_AlmAck"(Ib_CmdAck := #b_RstAlm,
	                 Oi_StaAlm => #i_dummy,
	                 Ob_StaAlm => #b_dummy,
	                 Ob_StaNewAlm => #b_StaAlmNew,
	                 IO_Alm0 := #b_AlmtoFb,
	                 IO_Alm1 := #b_Failure,
	                 IO_Alm2 := #b_NoAlm,
	                 IO_Alm3 := #b_NoAlm,
	                 IO_Alm4 := #b_NoAlm,
	                 IO_Alm5 := #b_NoAlm,
	                 IO_Alm6 := #b_NoAlm,
	                 IO_Alm7 := #b_NoAlm,
	                 IO_Alm8 := #b_NoAlm,
	                 IO_Alm9 := #b_NoAlm,
	                 IO_Alm10 := #b_NoAlm,
	                 IO_Alm11 := #b_NoAlm,
	                 IO_Alm12 := #b_NoAlm,
	                 IO_Alm13 := #b_NoAlm,
	                 IO_Alm14 := #b_NoAlm,
	                 IO_Alm15 := #b_NoAlm,
	                 IOi_StaAck := #i_AlmAck);

	// =============================================================================================================================
	//Failure Verification (Time-out feedback)
	IF (#Ii_ParTFb > 0) THEN  // only when time value > 0
	    #FB_UTIL_TON_Del_1(Ii_tValue := #Ii_ParTFb,
	                       Ib_In := (#b_CmdReqStart AND NOT #b_Running AND NOT #b_FbSimStart),
	                       Ii_Base := 1,
	                       Ib_Hold := 0,
	                       Ob_Out => #b_FbErrRun);
	END_IF;

	IF #Ib_Sta_Fail AND NOT #b_StaSim THEN  //Fault signal coming from machine
	    #b_Failure := TRUE;
	END_IF;

	IF  #b_FbErrRun AND #Ii_ParTFb > 0 AND NOT #b_DisAlmWrn AND NOT #b_StaSim THEN  //Fault feedback time out
	    #b_AlmtoFb := TRUE;
	END_IF;

	#b_StaAlm := #b_Failure OR #b_AlmtoFb;
	#Ob_StaAlm := #b_StaAlm;

	// =============================================================================================================================
	//HMI Status bits
	#Odi_HmiSta.%X0 := #b_StaModAut;
	#Odi_HmiSta.%X1 := #b_StaModMan;
	#Odi_HmiSta.%X2 := #b_StaModDis;
	#Odi_HmiSta.%X3 := #b_StaSim;               //Eqp in Simulation mode
	#Odi_HmiSta.%X4 := #b_StaIlOn;              //Eqp interlocked
	#Odi_HmiSta.%X5 := ((#b_Running AND NOT #b_StaSim) OR #b_FbSimStart) AND NOT #b_General_Purpouse AND NOT #b_StaIlOn;  //Status feedback on
	#Odi_HmiSta.%X6 := #b_StaAlm;               //Eqp alarm activated
	#Odi_HmiSta.%X7 := (#b_Running OR #b_FbSimStart) AND #b_General_Purpouse AND NOT #b_StaAlm; //Used for a general HMI animation
	#Odi_HmiSta.%X8 := ((#b_StaSim AND #b_FbSimStart) OR (NOT #b_StaSim AND #Ib_StaEqp1)) AND NOT #b_StaIlOn; //Status feedback Eqp1
	#Odi_HmiSta.%X9 := ((#b_StaSim AND #b_FbSimStart) OR (NOT #b_StaSim AND #Ib_StaEqp2)) AND NOT #b_StaIlOn; //Status feedback Eqp1

	// =============================================================================================================================
	//HMI Alarms bit
	#di_AUX := 0;
	#di_AUX.%X0 := #b_AlmtoFb;  //Feedback time out error
	#di_AUX.%X1 := #b_Failure;  //Machine signal error
	#di_AUX.%X2 := #Ib_ErrorEqp1 OR #b_StaAlm; //Eqp 1 Error
	#di_AUX.%X3 := #Ib_ErrorEqp2 OR #b_StaAlm; //Eqp 2 Error

	#Oi_HmiAlm := #di_AUX;

	// =============================================================================================================================

	//IO Area Feedback
	IF #b_StaModDis THEN
	    #IO_AreaFb.Mode.Dis := TRUE;
	END_IF;
	IF #b_StaModMan THEN
	    #IO_AreaFb.Mode.Man := TRUE;
	END_IF;
	IF #b_StaModAut THEN
	    #IO_AreaFb.Mode.Auto := TRUE;
	END_IF;
	IF #b_StaAlm THEN
	    #IO_AreaFb.Alm.Alm := TRUE;
	END_IF;
	IF #b_StaAlmNew THEN
	    #IO_AreaFb.Alm.New := TRUE;
	END_IF;
	IF #b_StaSim THEN
	    #IO_AreaFb.Sim.Sim := TRUE;
	END_IF;

	// =============================================================================================================================

	//Machine start-up counter
	IF (#Ob_StartReq AND #b_Running AND NOT #b_Old_Ob_Run) THEN
	    #Odi_ActCouRst := #Odi_ActCouRst + 1;
	    #Odi_ActCouTot := #Odi_ActCouTot + 1;
	END_IF;
	IF #b_HmiCmdRstActOpe THEN
	    #Odi_ActCouRst := 0;
	END_IF;

	#b_Old_Ob_Run := #Ob_StartReq;

	//Machine Time Operation
	#FB_UTIL_Work_H_Rst(Ib_On := #Ob_StartReq,
	                    Ib_Reset := #b_HmiCmdRstActOpe,
	                    Ib_Pls1S := "Clock_1Hz",
	                    IOdi_ResultHours := #Odi_RunTimRst);

	#FB_UTIL_Work_H_Tot(Ib_On := #Ob_StartReq,
	                    Ib_Pls1S := "Clock_1Hz",
	                    IOdi_ResultHours := #Odi_RunTimTot);

END_FUNCTION_BLOCK

FUNCTION_BLOCK "FB_Freq_Drive"
{ S7_Optimized_Access := 'FALSE' }
VERSION : 0.1
   VAR_INPUT
      Ir_SpOut : Real;   // Control output ACM
      Ir_ParMaxSpd : Real;   // Maximum speed
      Ir_ParMinSpd : Real;   // Minimum speed
      Ir_ParMaxRaw : Real;   // Maximum value for analog output mode
      Ir_ParMinRaw : Real;   // Minimum value for analog output mode
      Ib_Fwd : Bool;   // Control output forward ACM
      Ib_Off : Bool;   // Control output off ACM
      Ib_Reset : Bool;   // Reset alarms
      Ib_LocRem : Bool := TRUE;   // Control with PLC =1, Control local = 0
      Iw_Input : Word;   // First inputword of the drive
      Iw_Output : Word;   // First outputword of the drive
   END_VAR

   VAR_OUTPUT
      Or_ActSpd : Real;   // Actual speed drive
      Ob_FbFwd : Bool;   // Feedback forward
      Or_MotorCurrent : Real;   // Driver Actual Current
      Ob_FbLocGenEnab : Bool;   // Local General Enable
      Ob_FbDrwTest : Bool;   // Feedback Drawer in Test Position
      Ob_FbDrwInst : Bool;   // Feedback Drawer in Insert Position
      Ob_FbEmer : Bool;   // Feedback Emergency Button
      Oi_CurrentFault : Int;   // Driver Current Fault Number
      Ob_FbRem : Bool;   // Feedback CFW11 in Remote Mode
      Ob_CommFault : Bool;   // Communication Fault signal
   END_VAR

   VAR
      w_SpRaw : Word;
      r_SpRaw : Real;
      w_STW1 : Word;
      w_Status : Word;
      w_ActSpd : Word;
      r_ActSpd : Real;
      w_DriverCurrent : Word := 16#00;
      w_DriverFault : Word;
      I_DriveCurrent : Int := 16#0;
      R_DriveCurrent : Real;
      R_MotorActCurrent : Real;
      w_DIStatus : Word;
      b_FbLocGenEnab : Bool;   // Local General Enable
      b_FbDrwTest : Bool;   // Feedback Drawer in Test Position
      b_FbDrwInst : Bool;   // Feedback Drawer in Insert Position
      b_FbEmer : Bool;   // Feedback Emergency Button
      b_FbDI5Spare : Bool;   // Feedback DI 5 - Spare
      b_FbDI6Spare : Bool;   // Feedback DI 6 - Spare
      b_FbRem : Bool;   // Feedback CFW11 in Remote Mode
   END_VAR


BEGIN
	// =============================================================================================================================
	// Purpose: Reditech standard typical for controlling a frequency drive with Profibus
	// -----------------------------------------------------------------------------------------------------------------------------
	// Date (dd MMM yyyy)   Developer                   Version Comments/Reason for change
	// ..................   .........                   ....... ..........................
	// 06 nov 2018          Matthias De Staelen         01      Initial frequency drive control (creation)
	// 06 Dec 2019          Ivan Galhardoni             02      Code changed to control a WEG CFW11 freq. conv. model
	//
	// --------------------------------------------------- Initial AXM Release  ----------------------------------------------------
	// =============================================================================================================================
	//
	// Read inputwords drive
	#w_Status := PEEK_WORD(area := 16#81, dbNumber := 0, byteOffset := #Iw_Input);
	#w_ActSpd := PEEK_WORD(area := 16#81, dbNumber := 0, byteOffset := #Iw_Input + 2);
	#w_DriverCurrent := PEEK_WORD(area := 16#81, dbNumber := 0, byteOffset := #Iw_Input + 4);
	#w_DriverFault := PEEK_WORD(area := 16#81, dbNumber := 0, byteOffset := #Iw_Input + 6);
	#w_DIStatus := PEEK_WORD(area := 16#81, dbNumber := 0, byteOffset := #Iw_Input + 8);

	//Calculating the current motor speed and linearizing
	#r_ActSpd := DINT_TO_REAL(WORD_TO_DINT(#w_ActSpd));
	#Or_ActSpd := (((#r_ActSpd - #Ir_ParMinRaw) / (#Ir_ParMaxRaw - #Ir_ParMinRaw)) * (#Ir_ParMaxSpd - #Ir_ParMinSpd)) + #Ir_ParMinSpd;

	// Get feedback and alarm from statusword
	#Ob_FbFwd := #w_Status.%X8; //FeedbackRUN
	#Ob_CommFault := NOT #w_Status.%X9; //Communication Fault - Driver nor ready for receive command from DCS or Master (Always 1)
	#b_FbRem := #w_Status.%X12; //Feedback Remote Mode
	#Oi_CurrentFault := WORD_TO_INT(IN := #w_DriverFault);

	// Get information from DI
	#b_FbLocGenEnab := #w_DIStatus.%X0;
	#b_FbDrwTest := #w_DIStatus.%X1;
	#b_FbDrwInst := #w_DIStatus.%X2;
	#b_FbEmer := #w_DIStatus.%X3;
	#b_FbDI5Spare := #w_DIStatus.%X4;
	#b_FbDI6Spare := #w_DIStatus.%X5;

	#Ob_FbLocGenEnab := #b_FbLocGenEnab;
	#Ob_FbDrwTest := #b_FbDrwTest;
	#Ob_FbDrwInst := #b_FbDrwInst;
	#Ob_FbEmer := #b_FbEmer;
	#Ob_FbRem := #b_FbRem;

	//Calculating the Motor Current (Added by Jose Maximo)
	#I_DriveCurrent := WORD_TO_INT(#w_DriverCurrent);
	#R_DriveCurrent := INT_TO_REAL(#I_DriveCurrent);
	#R_MotorActCurrent := (#R_DriveCurrent / 10);
	#Or_MotorCurrent := #R_MotorActCurrent;

	// Calculating output
	#r_SpRaw := ((((#Ir_SpOut - #Ir_ParMinSpd) / (#Ir_ParMaxSpd - #Ir_ParMinSpd)) * (#Ir_ParMaxRaw - #Ir_ParMinRaw)) + #Ir_ParMinRaw);
	#w_SpRaw := INT_TO_WORD(IN := (REAL_TO_INT(IN := #r_SpRaw)));

	// Make the controlword for the drive (Changed By Jose Maximo)
	#w_STW1.%X0 := #Ib_Fwd AND NOT #Ib_Off; // Comando Gira/Pára Motor
	#w_STW1.%X1 := TRUE; // Habilita Geral
	#w_STW1.%X2 := TRUE; // Setido do Giro do Motor (Testar)
	#w_STW1.%X3 := FALSE;
	#w_STW1.%X4 := #Ib_LocRem;
	#w_STW1.%X5 := FALSE;
	#w_STW1.%X6 := FALSE;
	#w_STW1.%X7 := #Ib_Reset;

	// Write the information to the outputwords
	POKE(area:=16#82,
	     dbNumber:=0,
	     byteOffset:=#Iw_Output,
	     value:=#w_STW1);

	POKE(area := 16#82,
	     dbNumber := 0,
	     byteOffset := #Iw_Output + 2,
	     value := #w_SpRaw);

END_FUNCTION_BLOCK

FUNCTION_BLOCK "PID_CM_HMI"
{ S7_Optimized_Access := 'FALSE' }
VERSION : 0.1
   VAR_INPUT
      Ib_EnablePid : Bool;
      IO_AreaCmd : "UDT_AreaCmd";
      Ir_PvIn : Real;
      Ir_ParScMax : Real;
      Ir_ParScMin : Real;
      Ir_OutParScMax : Real;
      Ir_OutParScMin : Real;
      Iw_Cfg : Word;
      Ib_Rst : Bool;
   END_VAR

   VAR_OUTPUT
      Oi_Op_Mode : Int;
      Or_PvInMax : Real;
      Or_PvInMin : Real;
      Or_OutScMax : Real;
      Or_OutScMin : Real;
      Ob_ChangePID_Mode : Bool;
   END_VAR

   VAR_IN_OUT
      Ir_ManualValue : Real;   // Manual value for PID output
      IOdi_HmiCmd : DInt;   // Hmi received command bits
      Ir_ProportionalGain : Real;   // Kp
      Ir_IntregativeTime : Real;   // Ti
      Ir_DerivativeTime : Real;   // Td
      Ir_AutSp : Real;   // Automatic set point
      IOr_PropotionalGain : Real;
      IOr_IntegrativeTime : Real;
      IOr_DerivativeTime : Real;
      Ob_InvertControl : Bool;
   END_VAR

   VAR
      Auto_Mode : Bool;
      Manual_Mode : Bool;
      Disabled_Mode : Bool;
      Or_PidValue : Real;
      Odi_HmiSta : DInt;
      Ob_Alm : Bool;
      Odi_HmiAlm : DInt;
      Ob_Rst : Bool;
      b_Engineering_Control : Bool;
   END_VAR


BEGIN
	//Author: Ivan Galhardoni
	//Date: 19/May/2020
	//Usage: Block used for HMI communicatoion and PID control interface

	#Auto_Mode := #IO_AreaCmd.Mode.Auto;
	#Manual_Mode := #IO_AreaCmd.Mode.Man;
	#Disabled_Mode := #IO_AreaCmd.Mode.Dis;

	IF NOT #b_Engineering_Control THEN
	    #Ob_ChangePID_Mode := FALSE; //Erasing the rising edge signal to change the PID mode

	    //Writing the Operation mode to the PID controller
	    IF #Auto_Mode THEN
	        #Oi_Op_Mode := 3;
	        #Ir_ManualValue := 0.0;
	    END_IF;

	    IF #Manual_Mode THEN
	        #Oi_Op_Mode := 4;
	    END_IF;

	    IF #Disabled_Mode THEN
	        #Oi_Op_Mode := 0;
	        #Ir_ManualValue := 0.0;
	    END_IF;

	    //Scaling the PID controller input and output according to the controlled variable
	    #Or_PvInMax := #Ir_ParScMax;
	    #Or_PvInMin := #Ir_ParScMin;
	    #Or_OutScMax := #Ir_OutParScMax;
	    #Or_OutScMin := #Ir_OutParScMin;

	    //Selecting the controller direction type (Inverted or Direct)
	    #Ob_InvertControl := #Iw_Cfg.%X0;

	    //Preparing the PID controller constants
	    IF #IOdi_HmiCmd.%X2 THEN
	        #IOr_PropotionalGain := #Ir_ProportionalGain;
	        #IOr_IntegrativeTime := #Ir_IntregativeTime;
	        #IOr_DerivativeTime := #Ir_DerivativeTime;
	    END_IF;



	    IF #Oi_Op_Mode <> #Odi_HmiSta THEN

	        IF #Oi_Op_Mode = 0 AND #Odi_HmiSta <> 0 THEN
	            #Ob_ChangePID_Mode := TRUE;
	        END_IF;

	        IF #Oi_Op_Mode = 4 AND #Odi_HmiSta <> 4 THEN
	            #Ob_ChangePID_Mode := TRUE;
	        END_IF;

	    END_IF;

	    IF #Oi_Op_Mode = 3 AND #Ib_EnablePid AND #Odi_HmiSta <> 3 THEN
	        #Ob_ChangePID_Mode := TRUE;
	    ELSIF #Oi_Op_Mode = 3 AND NOT #Ib_EnablePid AND #Odi_HmiSta = 3 THEN
	        #Ob_ChangePID_Mode := TRUE;
	        #Oi_Op_Mode := 0;
	    END_IF;





	    //If there is an alarm, set up output alarm boolean
	    IF #Odi_HmiAlm > 0 THEN
	        #Ob_Alm := TRUE;
	    ELSE
	        #Ob_Alm := FALSE;
	    END_IF;

	    #Ob_Rst := #Ib_Rst OR #IOdi_HmiCmd.%X1; //Reset the PID controller block

	(* Hmi command bits must be reset at the end of the routine *)
	END_IF;
END_FUNCTION_BLOCK


FUNCTION_BLOCK "FB_CM_ACM"
TITLE = FB_AXV
{ S7_Optimized_Access := 'FALSE' }
AUTHOR : Reditech
FAMILY : Typicals
NAME : FB_AXV
VERSION : 0.1
//analog valve control
   VAR_INPUT
      Ib_AutFwd { ExternalVisible := 'False'} : Bool;   // automatic command forward
      Ib_AutRev { ExternalVisible := 'False'} : Bool;   // automatic command reversed
      Ib_FbFwd { ExternalVisible := 'False'} : Bool;   // feedback forward
      Ib_FbRev { ExternalVisible := 'False'} : Bool;   // feedback reversed
      ib_Is { ExternalVisible := 'False'} : Bool;   // Status Isolation switch (0=ok, 1=error)
      Ib_Mps { ExternalVisible := 'False'} : Bool;   // Status motor protection switch (0=ok, 1 = error)
      Ib_DevFlt : Bool;   // Hardware driver communication fault
      Ib_AlarmES : Bool;   // Driver Emergency stop button pressed
      Ib_DrawerInserted : Bool;   // Driver drawer inserted
      Ib_DrawerInTest : Bool;   // Driver drawer in test position
      Ib_Remote_Mode : Bool;   // Driver in Remote
      Ib_OverVoltage : Bool;   // Driver over voltage alarm
      Iby_Saf { ExternalVisible := 'False'} : Byte;   // 8 safety bits : 1=error
      Iby_IlFwd { ExternalVisible := 'False'} : Byte;   // 8 interlock bits : 1 prevents run forward
      Iby_IlRev { ExternalVisible := 'False'} : Byte;   // 8 interlock bits : 1 prevents run reverse
      Ib_Pls1S : Bool;
      Ir_ActSpd : Real;   // Actual speed (measurement)
      Ir_ParMaxSpd : Real;   // Maximum speed
      Ir_ParMinSpd : Real;   // Minimum speed
      Ir_ParCtlDev : Real;   // Control deviation (for digital output and feedback OK)
      Ir_ParMaxRaw : Real;   // Max value for analogue output mode
      Ir_ParMinRaw : Real;   // Min value for analogue output mode
      Ir_ParSafSpd : Real;   // Safety speed
      Ii_ParTO : Int;   // time out value for speed feedback monitoring
      Ii_ParTFb : Int;   // time out value for fwd or rev feedback monitoring
      Ii_ParTToRun : Int;   // time out value for time out run
      Ib_DisAlmWrn : Bool;
      Iw_Cfg { ExternalVisible := 'False'} : Word := 1;   // .0=analog pos present / .1=digital pos present
   END_VAR

   VAR_OUTPUT
      Or_SpOut : Real;   // Control output
      Ow_SpRaw : Word;   // Control output recalculated for analog output node
      Ob_Fwd { ExternalVisible := 'False'} : Bool;   // control output forward
      Ob_Rev { ExternalVisible := 'False'} : Bool;   // control output reverse
      Ob_Off { ExternalVisible := 'False'} : Bool := TRUE;   // control output off
      Ob_StaFwd : Bool;   // Status forward running
      Ob_StaRev : Bool;   // Status reverse running
      Ob_StaOff : Bool := TRUE;   // Status Off (not running)
      Ob_SpdOk { ExternalVisible := 'False'} : Bool;   // speed reached
      Or_StaSpd : Real;
      Ob_Alm { ExternalVisible := 'False'} : Bool;   // general alarm
      Ob_Wrn : Bool;   // general warning
      Odi_HmiSta : DInt;   // State bits for HMI
      Oi_HmiStaInd : DInt;
      Odi_HmiAlm : DInt;   // Alarm bit for HMI
      Odi_ActCouRst : DInt := 0;   // Actuation counter from last reset
      Odi_ActCouTot : DInt := 0;   // Total actuation counter
      Odi_RunTimRst : DInt;   // Operating hours from last reset
      Odi_RunTimTot : DInt;   // Total operating hours
      Oi_HmiAlm : Int;   // Pure alarm bits for HMI
      Ow_DCSSta : Word;
   END_VAR

   VAR_IN_OUT
      IOdi_HmiCmd : DInt;   // Command bits from HMI
      IOr_ManSP : Real;   // manual setpoint
      IOr_AutSp : Real;   // automatic setpoint
      IOr_SimSpd : Real;   // Simulated speed
      IO_AreaCmd : "UDT_AreaCmd";   // Command bits from area
      IO_AreaFb : "UDT_AreaFb";   // Feedback bits to area
   END_VAR

